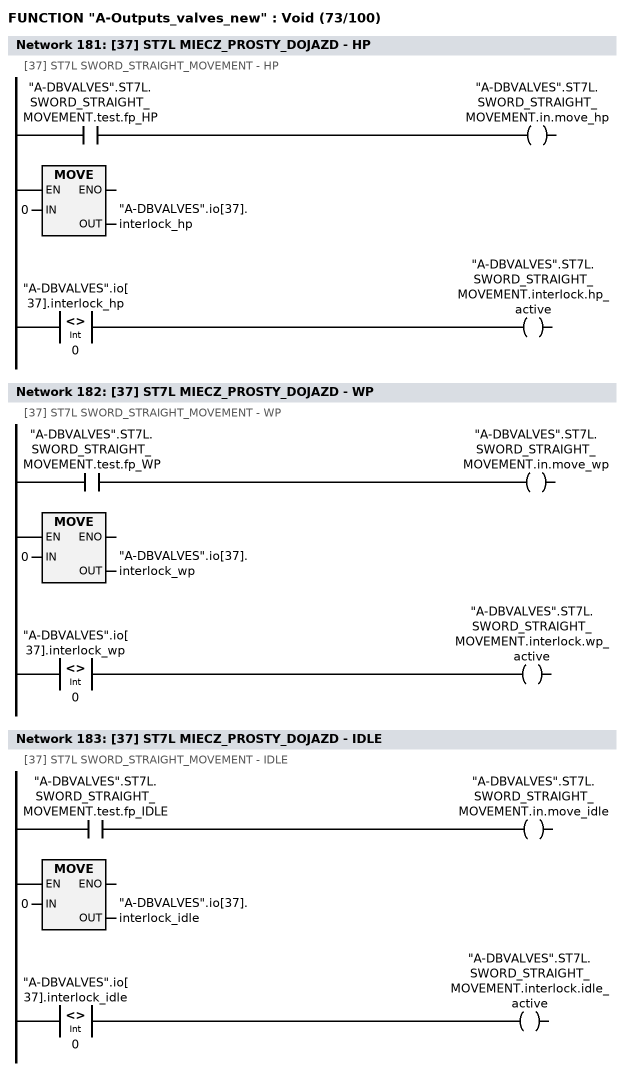
      O "A-DBVALVES".ST7L.SWORD_STRAIGHT_MOVEMENT.test.fp_HP;
//    O     "A-Flags".STATION.IN_HP_STEP
      = "A-DBVALVES".ST7L.SWORD_STRAIGHT_MOVEMENT.in.move_hp;

// Interlock hp
      L 0;
      T "A-DBVALVES".io[37].interlock_hp;

//{INTERLOCK_HP37}

      A(;
      L "A-DBVALVES".io[37].interlock_hp;
      L 0;
      <>I;
      );
      = "A-DBVALVES".ST7L.SWORD_STRAIGHT_MOVEMENT.interlock.hp_active;
NETWORK
TITLE = [37] ST7L MIECZ_PROSTY_DOJAZD - WP
//[37] ST7L SWORD_STRAIGHT_MOVEMENT - WP
      O "A-DBVALVES".ST7L.SWORD_STRAIGHT_MOVEMENT.test.fp_WP;
      = "A-DBVALVES".ST7L.SWORD_STRAIGHT_MOVEMENT.in.move_wp;

// Interlock wp
      L 0;
      T "A-DBVALVES".io[37].interlock_wp;

//{INTERLOCK_WP37}

      A(;
      L "A-DBVALVES".io[37].interlock_wp;
      L 0;
      <>I;
      );
      = "A-DBVALVES".ST7L.SWORD_STRAIGHT_MOVEMENT.interlock.wp_active;
NETWORK
TITLE = [37] ST7L MIECZ_PROSTY_DOJAZD - IDLE
//[37] ST7L SWORD_STRAIGHT_MOVEMENT - IDLE
      O "A-DBVALVES".ST7L.SWORD_STRAIGHT_MOVEMENT.test.fp_IDLE;
      = "A-DBVALVES".ST7L.SWORD_STRAIGHT_MOVEMENT.in.move_idle;

// Interlock idle
      L 0;
      T "A-DBVALVES".io[37].interlock_idle;

//{INTERLOCK_IDLE37}

      A(;
      L "A-DBVALVES".io[37].interlock_idle;
      L 0;
      <>I;
      );
      = "A-DBVALVES".ST7L.SWORD_STRAIGHT_MOVEMENT.interlock.idle_active;
NETWORK
TITLE = [37] ST7L MIECZ_PROSTY_DOJAZD
//[37] ST7L SWORD_STRAIGHT_MOVEMENT
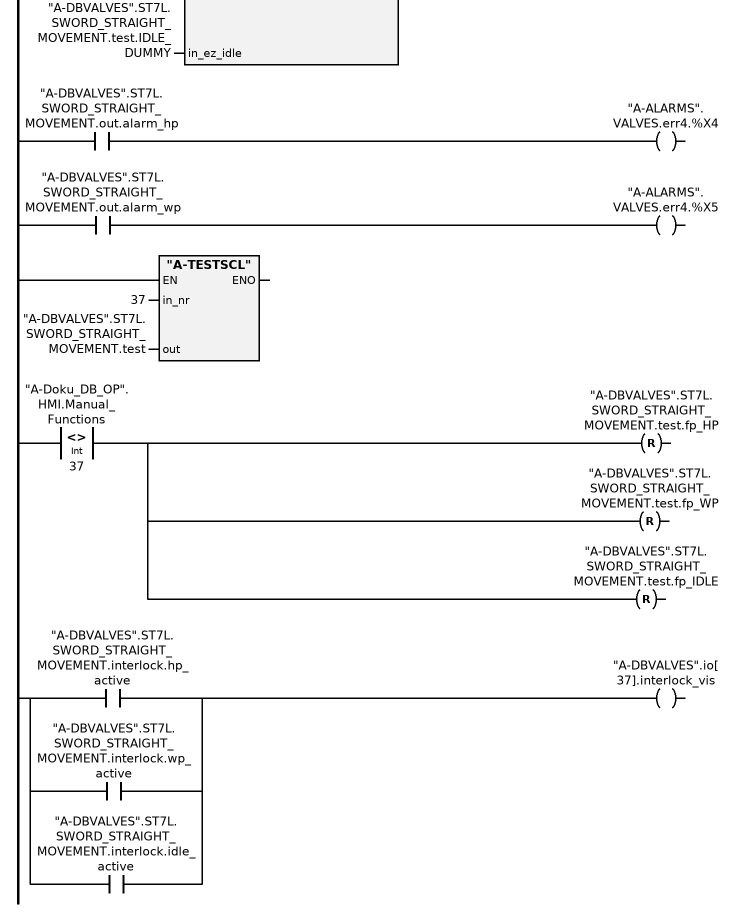
      CALL "3STATE_PISTON_with_brake", "INST_ST7L MIECZ_PROSTY_DOJAZD"
      (  in_safety_on                := "A-Flags".STATION.SAFETY_OK ,
         in_curtain_on               := "A-Flags".STATION.CURTAIN.OK ,
         in_move_hp                  := "A-DBVALVES".ST7L.SWORD_STRAIGHT_MOVEMENT.in.move_hp ,
         in_move_wp                  := "A-DBVALVES".ST7L.SWORD_STRAIGHT_MOVEMENT.in.move_wp ,
         in_move_idle                := "A-DBVALVES".ST7L.SWORD_STRAIGHT_MOVEMENT.in.move_idle ,
         in_interlock_hp             := "A-DBVALVES".ST7L.SWORD_STRAIGHT_MOVEMENT.interlock.hp_active ,
         in_interlock_wp             := "A-DBVALVES".ST7L.SWORD_STRAIGHT_MOVEMENT.interlock.wp_active ,
         in_interlock_idle           := "A-DBVALVES".ST7L.SWORD_STRAIGHT_MOVEMENT.interlock.idle_active ,
         in_sensor_hp1               := "ST7L-vsen_sword_straight_movement_HP_right" ,
         in_sensor_hp2               := "ST7L-vsen_sword_straight_movement_HP_right" ,
         in_sensor_wp1               := "ST7L-vsen_sword_straight_movement_WP_front" ,
         in_sensor_wp2               := "ST7L-vsen_sword_straight_movement_WP_front" ,
         out_in_hp                   := "A-DBVALVES".ST7L.SWORD_STRAIGHT_MOVEMENT.out.in_hp ,
         out_in_wp                   := "A-DBVALVES".ST7L.SWORD_STRAIGHT_MOVEMENT.out.in_wp ,
         out_idle                    := "A-DBVALVES".ST7L.SWORD_STRAIGHT_MOVEMENT.out.in_idle ,
         out_status                  := "A-DBVALVES".ST7L.SWORD_STRAIGHT_MOVEMENT.out.status ,
         out_brake                   := #brake ,
         out_alarm_hp                := "A-DBVALVES".ST7L.SWORD_STRAIGHT_MOVEMENT.out.alarm_hp ,
         out_alarm_wp                := "A-DBVALVES".ST7L.SWORD_STRAIGHT_MOVEMENT.out.alarm_wp ,
         out_alarm_idle              := "A-DBVALVES".ST7L.SWORD_STRAIGHT_MOVEMENT.out.alarm_idle ,
         out_diag_status             := "A-DBVALVES".ST7L.SWORD_STRAIGHT_MOVEMENT.out.diag_status ,
         out_interlock_show          := "A-DBVALVES".ST7L.SWORD_STRAIGHT_MOVEMENT.interlock.active ,
         in_ez_hp                    := "ST7L-ez_sword_straight_movement_HP_right" ,
         in_ez_wp                    := "ST7L-ez_sword_straight_movement_WP_front" ,
         in_ez_idle                  := "A-DBVALVES".ST7L.SWORD_STRAIGHT_MOVEMENT.test.IDLE_DUMMY
      );

      CALL "3STATE_DIAG"
      (  in_diag_status              := "A-DBVALVES".ST7L.SWORD_STRAIGHT_MOVEMENT.out.diag_status ,
         in_Ipw1                     := 'I120.0' ,
         in_Ipw2                     := ' ' ,
         in_Ipr1                     := 'I121.0' ,
         in_Ipr2                     := ' ' ,
         in_Qpw                      := 'Q3008.1' ,
         in_Qpr                      := 'Q3008.0' ,
         in_tio                      := "A-DBVALVES".io[37]
      );

      A "A-DBVALVES".ST7L.SWORD_STRAIGHT_MOVEMENT.out.alarm_hp;
      = "A-ALARMS".VALVES.err4.%X4;

      A "A-DBVALVES".ST7L.SWORD_STRAIGHT_MOVEMENT.out.alarm_wp;
      = "A-ALARMS".VALVES.err4.%X5;

      CALL "A-TESTSCL"
      (  in_nr                       := 37 ,
         out                         := "A-DBVALVES".ST7L.SWORD_STRAIGHT_MOVEMENT.test
      );

      A(;
      L "A-Doku_DB_OP".HMI.Manual_Functions;
      L 37;
      <>I;
      );
      R "A-DBVALVES".ST7L.SWORD_STRAIGHT_MOVEMENT.test.fp_HP;
      R "A-DBVALVES".ST7L.SWORD_STRAIGHT_MOVEMENT.test.fp_WP;
      R "A-DBVALVES".ST7L.SWORD_STRAIGHT_MOVEMENT.test.fp_IDLE;

      O "A-DBVALVES".ST7L.SWORD_STRAIGHT_MOVEMENT.interlock.hp_active;
      O "A-DBVALVES".ST7L.SWORD_STRAIGHT_MOVEMENT.interlock.wp_active;
      O "A-DBVALVES".ST7L.SWORD_STRAIGHT_MOVEMENT.interlock.idle_active;
      = "A-DBVALVES".io[37].interlock_vis;
NETWORK
TITLE = -

NETWORK
TITLE = [38] ST7L MIECZ_PROSTY - HP
//[38] ST7L SWORD_STRAIGHT - HP
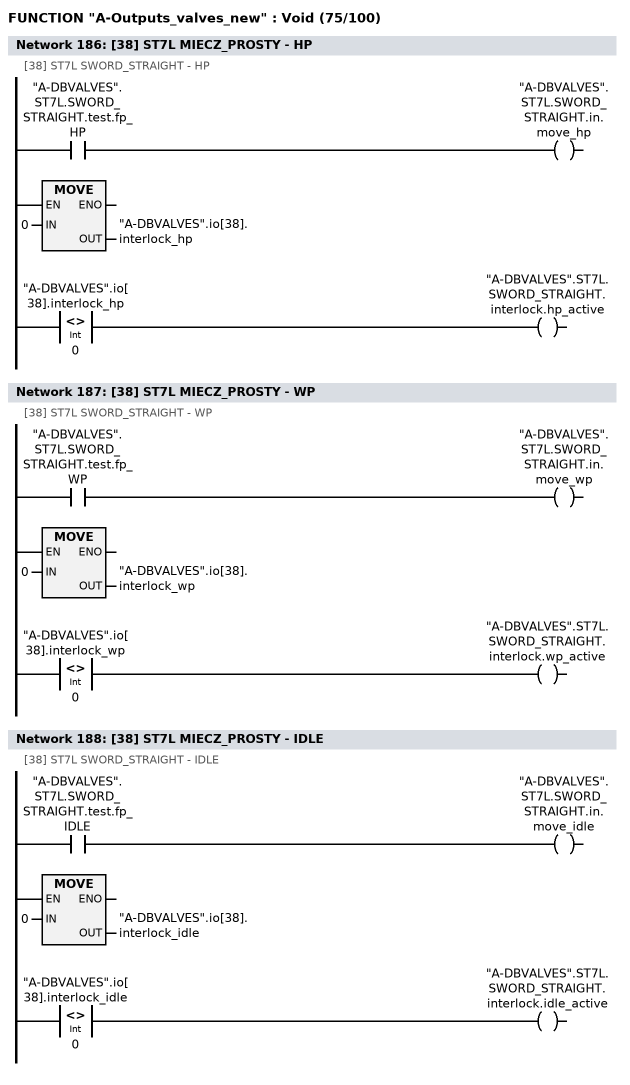
      O "A-DBVALVES".ST7L.SWORD_STRAIGHT.test.fp_HP;
//    O     "A-Flags".STATION.IN_HP_STEP
      = "A-DBVALVES".ST7L.SWORD_STRAIGHT.in.move_hp;

// Interlock hp
      L 0;
      T "A-DBVALVES".io[38].interlock_hp;

//{INTERLOCK_HP38}

      A(;
      L "A-DBVALVES".io[38].interlock_hp;
      L 0;
      <>I;
      );
      = "A-DBVALVES".ST7L.SWORD_STRAIGHT.interlock.hp_active;
NETWORK
TITLE = [38] ST7L MIECZ_PROSTY - WP
//[38] ST7L SWORD_STRAIGHT - WP
      O "A-DBVALVES".ST7L.SWORD_STRAIGHT.test.fp_WP;
      = "A-DBVALVES".ST7L.SWORD_STRAIGHT.in.move_wp;

// Interlock wp
      L 0;
      T "A-DBVALVES".io[38].interlock_wp;

//{INTERLOCK_WP38}

      A(;
      L "A-DBVALVES".io[38].interlock_wp;
      L 0;
      <>I;
      );
      = "A-DBVALVES".ST7L.SWORD_STRAIGHT.interlock.wp_active;
NETWORK
TITLE = [38] ST7L MIECZ_PROSTY - IDLE
//[38] ST7L SWORD_STRAIGHT - IDLE
      O "A-DBVALVES".ST7L.SWORD_STRAIGHT.test.fp_IDLE;
      = "A-DBVALVES".ST7L.SWORD_STRAIGHT.in.move_idle;

// Interlock idle
      L 0;
      T "A-DBVALVES".io[38].interlock_idle;

//{INTERLOCK_IDLE38}

      A(;
      L "A-DBVALVES".io[38].interlock_idle;
      L 0;
      <>I;
      );
      = "A-DBVALVES".ST7L.SWORD_STRAIGHT.interlock.idle_active;
NETWORK
TITLE = [38] ST7L MIECZ_PROSTY
//[38] ST7L SWORD_STRAIGHT
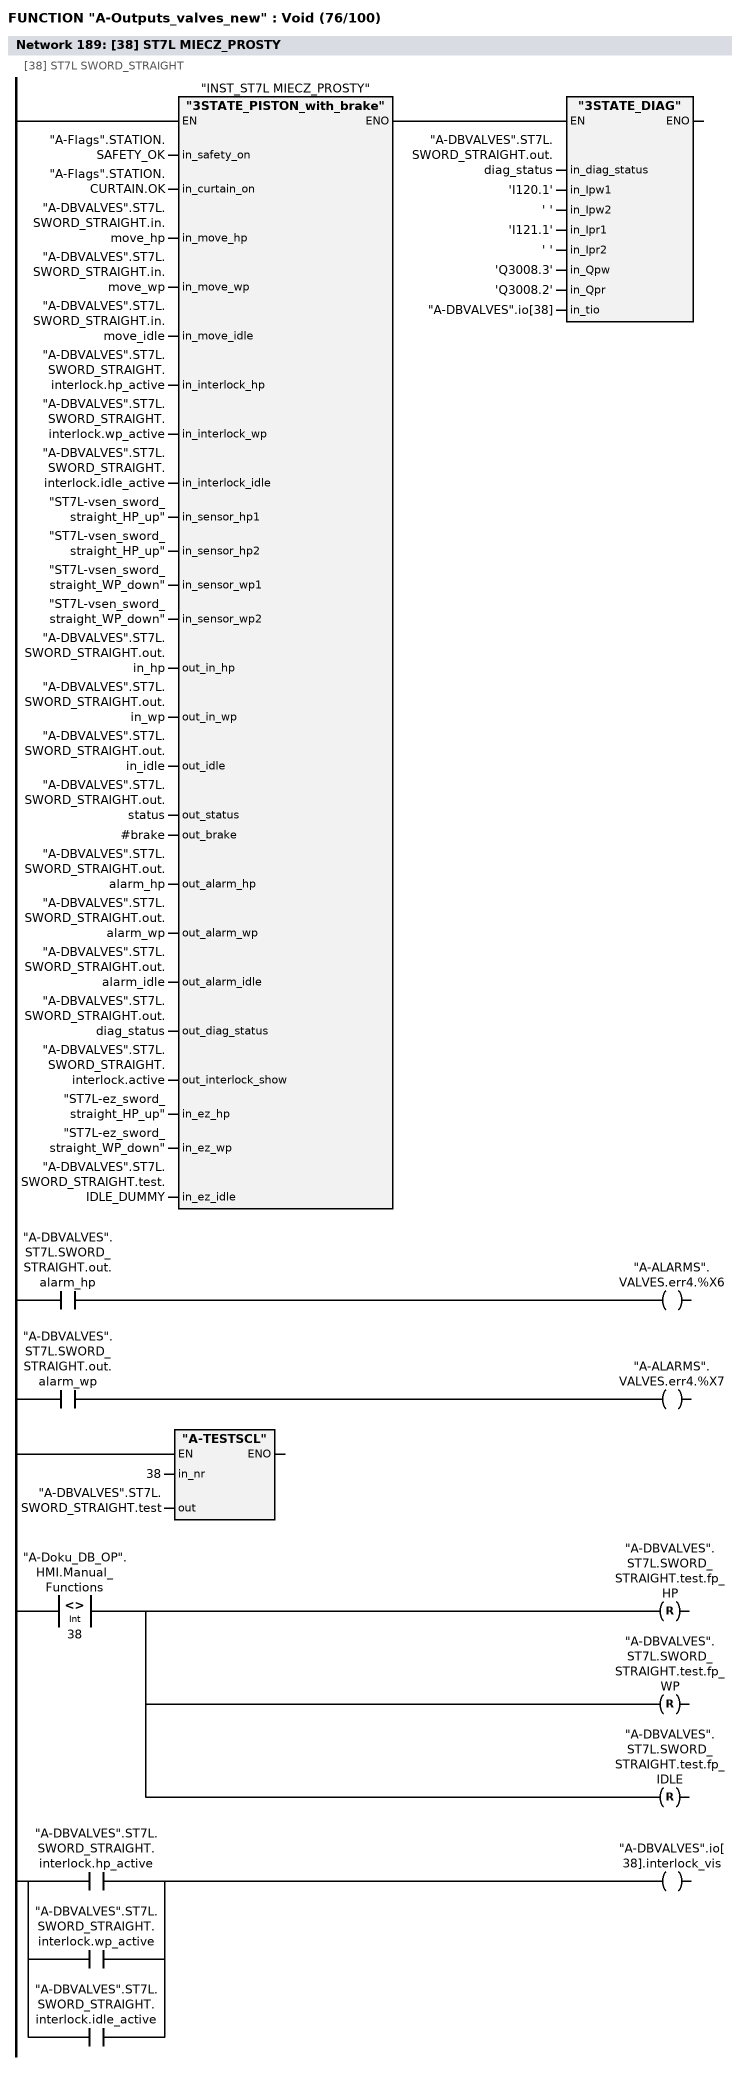
      CALL "3STATE_PISTON_with_brake", "INST_ST7L MIECZ_PROSTY"
      (  in_safety_on                := "A-Flags".STATION.SAFETY_OK ,
         in_curtain_on               := "A-Flags".STATION.CURTAIN.OK ,
         in_move_hp                  := "A-DBVALVES".ST7L.SWORD_STRAIGHT.in.move_hp ,
         in_move_wp                  := "A-DBVALVES".ST7L.SWORD_STRAIGHT.in.move_wp ,
         in_move_idle                := "A-DBVALVES".ST7L.SWORD_STRAIGHT.in.move_idle ,
         in_interlock_hp             := "A-DBVALVES".ST7L.SWORD_STRAIGHT.interlock.hp_active ,
         in_interlock_wp             := "A-DBVALVES".ST7L.SWORD_STRAIGHT.interlock.wp_active ,
         in_interlock_idle           := "A-DBVALVES".ST7L.SWORD_STRAIGHT.interlock.idle_active ,
         in_sensor_hp1               := "ST7L-vsen_sword_straight_HP_up" ,
         in_sensor_hp2               := "ST7L-vsen_sword_straight_HP_up" ,
         in_sensor_wp1               := "ST7L-vsen_sword_straight_WP_down" ,
         in_sensor_wp2               := "ST7L-vsen_sword_straight_WP_down" ,
         out_in_hp                   := "A-DBVALVES".ST7L.SWORD_STRAIGHT.out.in_hp ,
         out_in_wp                   := "A-DBVALVES".ST7L.SWORD_STRAIGHT.out.in_wp ,
         out_idle                    := "A-DBVALVES".ST7L.SWORD_STRAIGHT.out.in_idle ,
         out_status                  := "A-DBVALVES".ST7L.SWORD_STRAIGHT.out.status ,
         out_brake                   := #brake ,
         out_alarm_hp                := "A-DBVALVES".ST7L.SWORD_STRAIGHT.out.alarm_hp ,
         out_alarm_wp                := "A-DBVALVES".ST7L.SWORD_STRAIGHT.out.alarm_wp ,
         out_alarm_idle              := "A-DBVALVES".ST7L.SWORD_STRAIGHT.out.alarm_idle ,
         out_diag_status             := "A-DBVALVES".ST7L.SWORD_STRAIGHT.out.diag_status ,
         out_interlock_show          := "A-DBVALVES".ST7L.SWORD_STRAIGHT.interlock.active ,
         in_ez_hp                    := "ST7L-ez_sword_straight_HP_up" ,
         in_ez_wp                    := "ST7L-ez_sword_straight_WP_down" ,
         in_ez_idle                  := "A-DBVALVES".ST7L.SWORD_STRAIGHT.test.IDLE_DUMMY
      );

      CALL "3STATE_DIAG"
      (  in_diag_status              := "A-DBVALVES".ST7L.SWORD_STRAIGHT.out.diag_status ,
         in_Ipw1                     := 'I120.1' ,
         in_Ipw2                     := ' ' ,
         in_Ipr1                     := 'I121.1' ,
         in_Ipr2                     := ' ' ,
         in_Qpw                      := 'Q3008.3' ,
         in_Qpr                      := 'Q3008.2' ,
         in_tio                      := "A-DBVALVES".io[38]
      );

      A "A-DBVALVES".ST7L.SWORD_STRAIGHT.out.alarm_hp;
      = "A-ALARMS".VALVES.err4.%X6;

      A "A-DBVALVES".ST7L.SWORD_STRAIGHT.out.alarm_wp;
      = "A-ALARMS".VALVES.err4.%X7;

      CALL "A-TESTSCL"
      (  in_nr                       := 38 ,
         out                         := "A-DBVALVES".ST7L.SWORD_STRAIGHT.test
      );

      A(;
      L "A-Doku_DB_OP".HMI.Manual_Functions;
      L 38;
      <>I;
      );
      R "A-DBVALVES".ST7L.SWORD_STRAIGHT.test.fp_HP;
      R "A-DBVALVES".ST7L.SWORD_STRAIGHT.test.fp_WP;
      R "A-DBVALVES".ST7L.SWORD_STRAIGHT.test.fp_IDLE;

      O "A-DBVALVES".ST7L.SWORD_STRAIGHT.interlock.hp_active;
      O "A-DBVALVES".ST7L.SWORD_STRAIGHT.interlock.wp_active;
      O "A-DBVALVES".ST7L.SWORD_STRAIGHT.interlock.idle_active;
      = "A-DBVALVES".io[38].interlock_vis;
NETWORK
TITLE = -

NETWORK
TITLE = [39] ST7L MIECZ_RUCHOMY_DOJAZD - HP
//[39] ST7L SWORD_MOBILE_MOVEMENT - HP
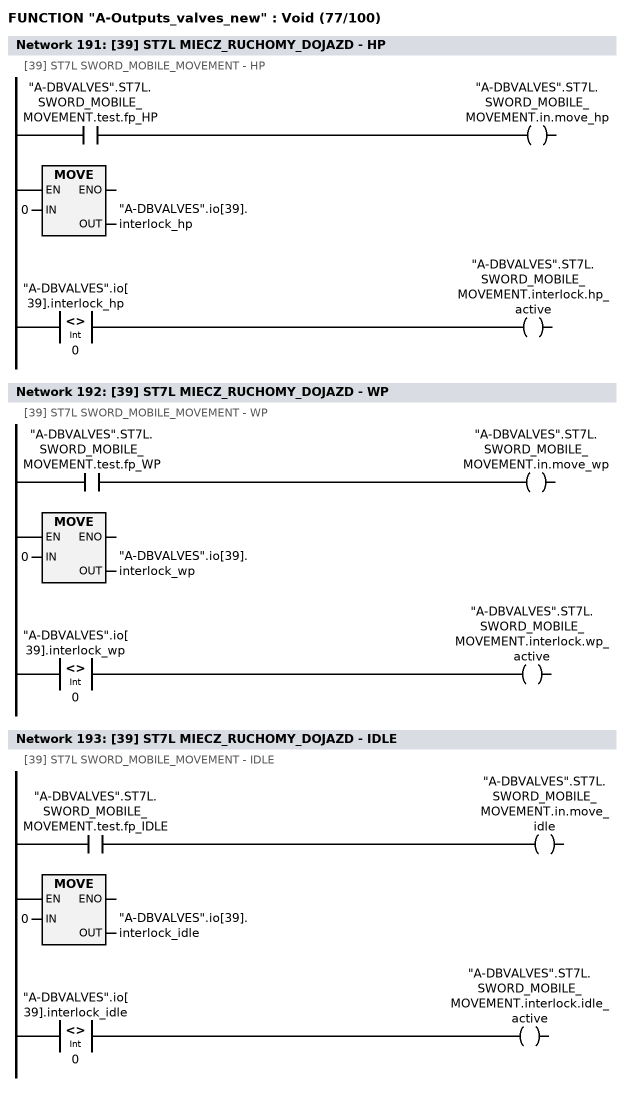
      O "A-DBVALVES".ST7L.SWORD_MOBILE_MOVEMENT.test.fp_HP;
//    O     "A-Flags".STATION.IN_HP_STEP
      = "A-DBVALVES".ST7L.SWORD_MOBILE_MOVEMENT.in.move_hp;

// Interlock hp
      L 0;
      T "A-DBVALVES".io[39].interlock_hp;

//{INTERLOCK_HP39}

      A(;
      L "A-DBVALVES".io[39].interlock_hp;
      L 0;
      <>I;
      );
      = "A-DBVALVES".ST7L.SWORD_MOBILE_MOVEMENT.interlock.hp_active;
NETWORK
TITLE = [39] ST7L MIECZ_RUCHOMY_DOJAZD - WP
//[39] ST7L SWORD_MOBILE_MOVEMENT - WP
      O "A-DBVALVES".ST7L.SWORD_MOBILE_MOVEMENT.test.fp_WP;
      = "A-DBVALVES".ST7L.SWORD_MOBILE_MOVEMENT.in.move_wp;

// Interlock wp
      L 0;
      T "A-DBVALVES".io[39].interlock_wp;

//{INTERLOCK_WP39}

      A(;
      L "A-DBVALVES".io[39].interlock_wp;
      L 0;
      <>I;
      );
      = "A-DBVALVES".ST7L.SWORD_MOBILE_MOVEMENT.interlock.wp_active;
NETWORK
TITLE = [39] ST7L MIECZ_RUCHOMY_DOJAZD - IDLE
//[39] ST7L SWORD_MOBILE_MOVEMENT - IDLE
      O "A-DBVALVES".ST7L.SWORD_MOBILE_MOVEMENT.test.fp_IDLE;
      = "A-DBVALVES".ST7L.SWORD_MOBILE_MOVEMENT.in.move_idle;

// Interlock idle
      L 0;
      T "A-DBVALVES".io[39].interlock_idle;

//{INTERLOCK_IDLE39}

      A(;
      L "A-DBVALVES".io[39].interlock_idle;
      L 0;
      <>I;
      );
      = "A-DBVALVES".ST7L.SWORD_MOBILE_MOVEMENT.interlock.idle_active;
NETWORK
TITLE = [39] ST7L MIECZ_RUCHOMY_DOJAZD
//[39] ST7L SWORD_MOBILE_MOVEMENT
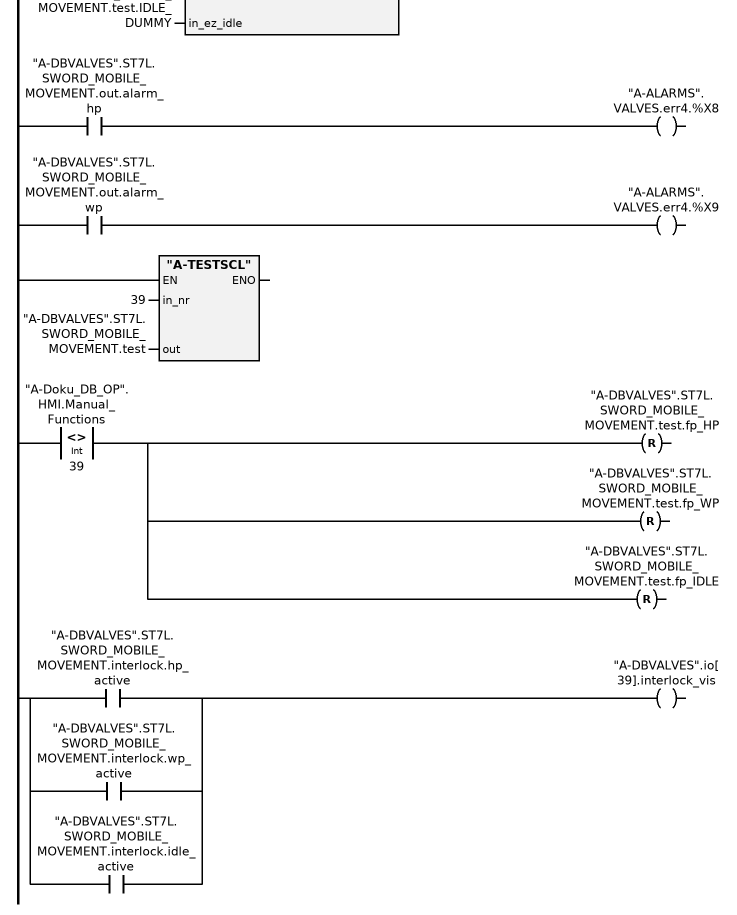
      CALL "3STATE_PISTON_with_brake", "INST_ST7L MIECZ_RUCHOMY_DOJAZD"
      (  in_safety_on                := "A-Flags".STATION.SAFETY_OK ,
         in_curtain_on               := "A-Flags".STATION.CURTAIN.OK ,
         in_move_hp                  := "A-DBVALVES".ST7L.SWORD_MOBILE_MOVEMENT.in.move_hp ,
         in_move_wp                  := "A-DBVALVES".ST7L.SWORD_MOBILE_MOVEMENT.in.move_wp ,
         in_move_idle                := "A-DBVALVES".ST7L.SWORD_MOBILE_MOVEMENT.in.move_idle ,
         in_interlock_hp             := "A-DBVALVES".ST7L.SWORD_MOBILE_MOVEMENT.interlock.hp_active ,
         in_interlock_wp             := "A-DBVALVES".ST7L.SWORD_MOBILE_MOVEMENT.interlock.wp_active ,
         in_interlock_idle           := "A-DBVALVES".ST7L.SWORD_MOBILE_MOVEMENT.interlock.idle_active ,
         in_sensor_hp1               := "ST7L-vsen_sword_mobile_movement_HP_right" ,
         in_sensor_hp2               := "ST7L-vsen_sword_mobile_movement_HP_right" ,
         in_sensor_wp1               := "ST7L-vsen_sword_mobile_movement_WP_front" ,
         in_sensor_wp2               := "ST7L-vsen_sword_mobile_movement_WP_front" ,
         out_in_hp                   := "A-DBVALVES".ST7L.SWORD_MOBILE_MOVEMENT.out.in_hp ,
         out_in_wp                   := "A-DBVALVES".ST7L.SWORD_MOBILE_MOVEMENT.out.in_wp ,
         out_idle                    := "A-DBVALVES".ST7L.SWORD_MOBILE_MOVEMENT.out.in_idle ,
         out_status                  := "A-DBVALVES".ST7L.SWORD_MOBILE_MOVEMENT.out.status ,
         out_brake                   := #brake ,
         out_alarm_hp                := "A-DBVALVES".ST7L.SWORD_MOBILE_MOVEMENT.out.alarm_hp ,
         out_alarm_wp                := "A-DBVALVES".ST7L.SWORD_MOBILE_MOVEMENT.out.alarm_wp ,
         out_alarm_idle              := "A-DBVALVES".ST7L.SWORD_MOBILE_MOVEMENT.out.alarm_idle ,
         out_diag_status             := "A-DBVALVES".ST7L.SWORD_MOBILE_MOVEMENT.out.diag_status ,
         out_interlock_show          := "A-DBVALVES".ST7L.SWORD_MOBILE_MOVEMENT.interlock.active ,
         in_ez_hp                    := "ST7L-ez_sword_mobile_movement_HP_right" ,
         in_ez_wp                    := "ST7L-ez_sword_mobile_movement_WP_front" ,
         in_ez_idle                  := "A-DBVALVES".ST7L.SWORD_MOBILE_MOVEMENT.test.IDLE_DUMMY
      );

      CALL "3STATE_DIAG"
      (  in_diag_status              := "A-DBVALVES".ST7L.SWORD_MOBILE_MOVEMENT.out.diag_status ,
         in_Ipw1                     := 'I120.3' ,
         in_Ipw2                     := ' ' ,
         in_Ipr1                     := 'I121.3' ,
         in_Ipr2                     := ' ' ,
         in_Qpw                      := 'Q3008.7' ,
         in_Qpr                      := 'Q3008.6' ,
         in_tio                      := "A-DBVALVES".io[39]
      );

      A "A-DBVALVES".ST7L.SWORD_MOBILE_MOVEMENT.out.alarm_hp;
      = "A-ALARMS".VALVES.err4.%X8;

      A "A-DBVALVES".ST7L.SWORD_MOBILE_MOVEMENT.out.alarm_wp;
      = "A-ALARMS".VALVES.err4.%X9;

      CALL "A-TESTSCL"
      (  in_nr                       := 39 ,
         out                         := "A-DBVALVES".ST7L.SWORD_MOBILE_MOVEMENT.test
      );

      A(;
      L "A-Doku_DB_OP".HMI.Manual_Functions;
      L 39;
      <>I;
      );
      R "A-DBVALVES".ST7L.SWORD_MOBILE_MOVEMENT.test.fp_HP;
      R "A-DBVALVES".ST7L.SWORD_MOBILE_MOVEMENT.test.fp_WP;
      R "A-DBVALVES".ST7L.SWORD_MOBILE_MOVEMENT.test.fp_IDLE;

      O "A-DBVALVES".ST7L.SWORD_MOBILE_MOVEMENT.interlock.hp_active;
      O "A-DBVALVES".ST7L.SWORD_MOBILE_MOVEMENT.interlock.wp_active;
      O "A-DBVALVES".ST7L.SWORD_MOBILE_MOVEMENT.interlock.idle_active;
      = "A-DBVALVES".io[39].interlock_vis;
NETWORK
TITLE = -

NETWORK
TITLE = [40] ST7L MIECZ_RUCHOMY_PRZEJAZD - HP
//[40] ST7L SWORD_MOBILE_SLIDE - HP
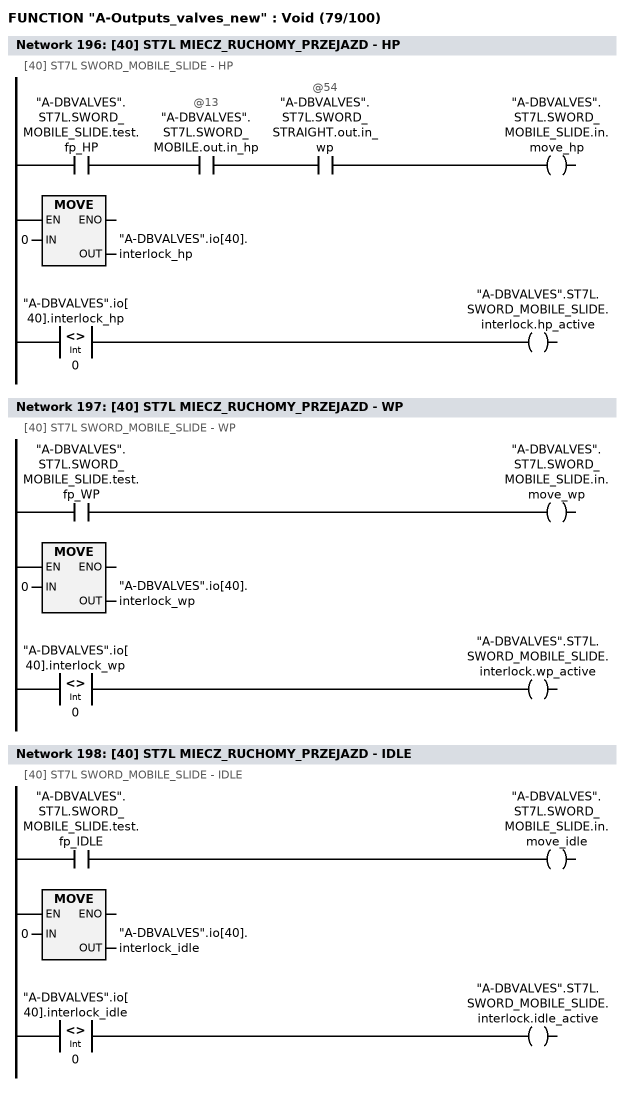
      O "A-DBVALVES".ST7L.SWORD_MOBILE_SLIDE.test.fp_HP;
//    O     "A-Flags".STATION.IN_HP_STEP
      A "A-DBVALVES".ST7L.SWORD_MOBILE.out.in_hp;// @13
      A "A-DBVALVES".ST7L.SWORD_STRAIGHT.out.in_wp;// @54
      = "A-DBVALVES".ST7L.SWORD_MOBILE_SLIDE.in.move_hp;

// Interlock hp
      L 0;
      T "A-DBVALVES".io[40].interlock_hp;

//{INTERLOCK_HP40}

      A(;
      L "A-DBVALVES".io[40].interlock_hp;
      L 0;
      <>I;
      );
      = "A-DBVALVES".ST7L.SWORD_MOBILE_SLIDE.interlock.hp_active;
NETWORK
TITLE = [40] ST7L MIECZ_RUCHOMY_PRZEJAZD - WP
//[40] ST7L SWORD_MOBILE_SLIDE - WP
      O "A-DBVALVES".ST7L.SWORD_MOBILE_SLIDE.test.fp_WP;
      = "A-DBVALVES".ST7L.SWORD_MOBILE_SLIDE.in.move_wp;

// Interlock wp
      L 0;
      T "A-DBVALVES".io[40].interlock_wp;

//{INTERLOCK_WP40}

      A(;
      L "A-DBVALVES".io[40].interlock_wp;
      L 0;
      <>I;
      );
      = "A-DBVALVES".ST7L.SWORD_MOBILE_SLIDE.interlock.wp_active;
NETWORK
TITLE = [40] ST7L MIECZ_RUCHOMY_PRZEJAZD - IDLE
//[40] ST7L SWORD_MOBILE_SLIDE - IDLE
      O "A-DBVALVES".ST7L.SWORD_MOBILE_SLIDE.test.fp_IDLE;
      = "A-DBVALVES".ST7L.SWORD_MOBILE_SLIDE.in.move_idle;

// Interlock idle
      L 0;
      T "A-DBVALVES".io[40].interlock_idle;

//{INTERLOCK_IDLE40}

      A(;
      L "A-DBVALVES".io[40].interlock_idle;
      L 0;
      <>I;
      );
      = "A-DBVALVES".ST7L.SWORD_MOBILE_SLIDE.interlock.idle_active;
NETWORK
TITLE = [40] ST7L MIECZ_RUCHOMY_PRZEJAZD
//[40] ST7L SWORD_MOBILE_SLIDE
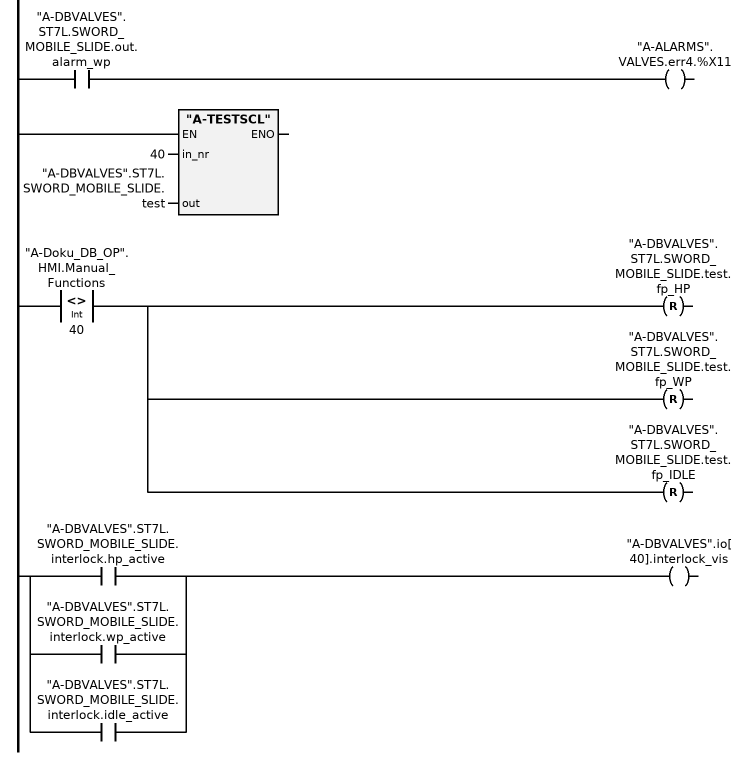
      CALL "3STATE_PISTON_with_brake", "INST_ST7L MIECZ_RUCHOMY_PRZEJAZD"
      (  in_safety_on                := "A-Flags".STATION.SAFETY_OK ,
         in_curtain_on               := "A-Flags".STATION.CURTAIN.OK ,
         in_move_hp                  := "A-DBVALVES".ST7L.SWORD_MOBILE_SLIDE.in.move_hp ,
         in_move_wp                  := "A-DBVALVES".ST7L.SWORD_MOBILE_SLIDE.in.move_wp ,
         in_move_idle                := "A-DBVALVES".ST7L.SWORD_MOBILE_SLIDE.in.move_idle ,
         in_interlock_hp             := "A-DBVALVES".ST7L.SWORD_MOBILE_SLIDE.interlock.hp_active ,
         in_interlock_wp             := "A-DBVALVES".ST7L.SWORD_MOBILE_SLIDE.interlock.wp_active ,
         in_interlock_idle           := "A-DBVALVES".ST7L.SWORD_MOBILE_SLIDE.interlock.idle_active ,
         in_sensor_hp1               := "ST7L-vsen_sword_mobile_slide_HP_left" ,
         in_sensor_hp2               := "ST7L-vsen_sword_mobile_slide_HP_left" ,
         in_sensor_wp1               := "ST7L-vsen_sword_mobile_slide_WP_right" ,
         in_sensor_wp2               := "ST7L-vsen_sword_mobile_slide_WP_right" ,
         out_in_hp                   := "A-DBVALVES".ST7L.SWORD_MOBILE_SLIDE.out.in_hp ,
         out_in_wp                   := "A-DBVALVES".ST7L.SWORD_MOBILE_SLIDE.out.in_wp ,
         out_idle                    := "A-DBVALVES".ST7L.SWORD_MOBILE_SLIDE.out.in_idle ,
         out_status                  := "A-DBVALVES".ST7L.SWORD_MOBILE_SLIDE.out.status ,
         out_brake                   := #brake ,
         out_alarm_hp                := "A-DBVALVES".ST7L.SWORD_MOBILE_SLIDE.out.alarm_hp ,
         out_alarm_wp                := "A-DBVALVES".ST7L.SWORD_MOBILE_SLIDE.out.alarm_wp ,
         out_alarm_idle              := "A-DBVALVES".ST7L.SWORD_MOBILE_SLIDE.out.alarm_idle ,
         out_diag_status             := "A-DBVALVES".ST7L.SWORD_MOBILE_SLIDE.out.diag_status ,
         out_interlock_show          := "A-DBVALVES".ST7L.SWORD_MOBILE_SLIDE.interlock.active ,
         in_ez_hp                    := "ST7L-ez_sword_mobile_slide_HP_left" ,
         in_ez_wp                    := "ST7L-ez_sword_mobile_slide_WP_right" ,
         in_ez_idle                  := "A-DBVALVES".ST7L.SWORD_MOBILE_SLIDE.test.IDLE_DUMMY
      );

      CALL "3STATE_DIAG"
      (  in_diag_status              := "A-DBVALVES".ST7L.SWORD_MOBILE_SLIDE.out.diag_status ,
         in_Ipw1                     := 'I120.2' ,
         in_Ipw2                     := ' ' ,
         in_Ipr1                     := 'I121.2' ,
         in_Ipr2                     := ' ' ,
         in_Qpw                      := 'Q3008.5' ,
         in_Qpr                      := 'Q3008.4' ,
         in_tio                      := "A-DBVALVES".io[40]
      );

      A "A-DBVALVES".ST7L.SWORD_MOBILE_SLIDE.out.alarm_hp;
      = "A-ALARMS".VALVES.err4.%X10;

      A "A-DBVALVES".ST7L.SWORD_MOBILE_SLIDE.out.alarm_wp;
      = "A-ALARMS".VALVES.err4.%X11;

      CALL "A-TESTSCL"
      (  in_nr                       := 40 ,
         out                         := "A-DBVALVES".ST7L.SWORD_MOBILE_SLIDE.test
      );

      A(;
      L "A-Doku_DB_OP".HMI.Manual_Functions;
      L 40;
      <>I;
      );
      R "A-DBVALVES".ST7L.SWORD_MOBILE_SLIDE.test.fp_HP;
      R "A-DBVALVES".ST7L.SWORD_MOBILE_SLIDE.test.fp_WP;
      R "A-DBVALVES".ST7L.SWORD_MOBILE_SLIDE.test.fp_IDLE;

      O "A-DBVALVES".ST7L.SWORD_MOBILE_SLIDE.interlock.hp_active;
      O "A-DBVALVES".ST7L.SWORD_MOBILE_SLIDE.interlock.wp_active;
      O "A-DBVALVES".ST7L.SWORD_MOBILE_SLIDE.interlock.idle_active;
      = "A-DBVALVES".io[40].interlock_vis;
NETWORK
TITLE = -

NETWORK
TITLE = [41] ST7L MIECZ_RUCHOMY - HP
//[41] ST7L SWORD_MOBILE - HP
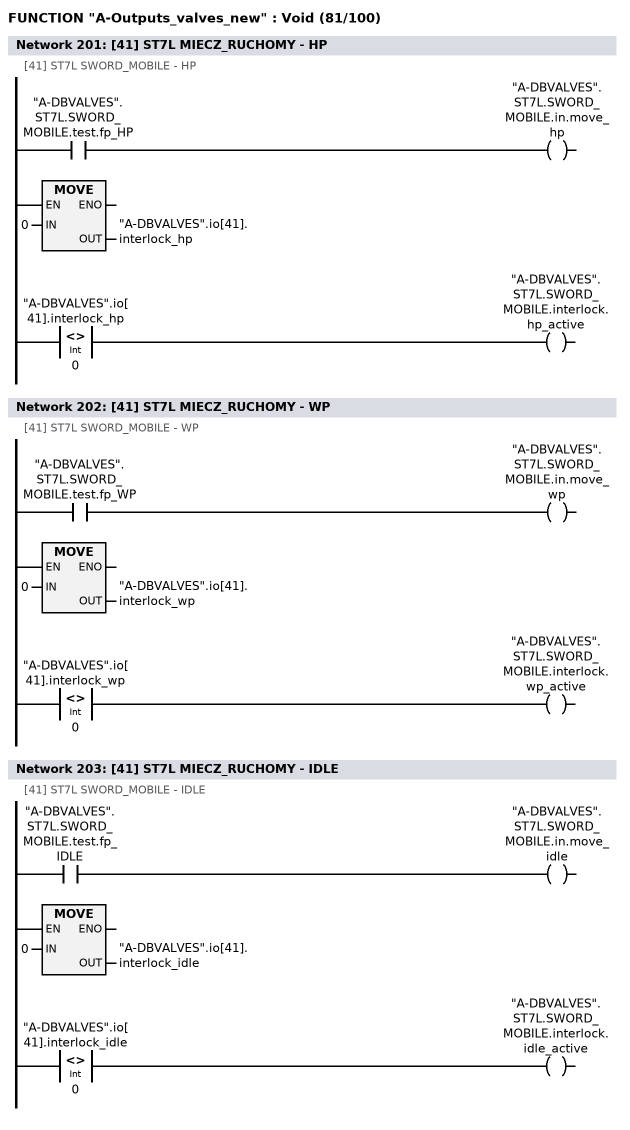
      O "A-DBVALVES".ST7L.SWORD_MOBILE.test.fp_HP;
//    O     "A-Flags".STATION.IN_HP_STEP
      = "A-DBVALVES".ST7L.SWORD_MOBILE.in.move_hp;

// Interlock hp
      L 0;
      T "A-DBVALVES".io[41].interlock_hp;

//{INTERLOCK_HP41}

      A(;
      L "A-DBVALVES".io[41].interlock_hp;
      L 0;
      <>I;
      );
      = "A-DBVALVES".ST7L.SWORD_MOBILE.interlock.hp_active;
NETWORK
TITLE = [41] ST7L MIECZ_RUCHOMY - WP
//[41] ST7L SWORD_MOBILE - WP
      O "A-DBVALVES".ST7L.SWORD_MOBILE.test.fp_WP;
      = "A-DBVALVES".ST7L.SWORD_MOBILE.in.move_wp;

// Interlock wp
      L 0;
      T "A-DBVALVES".io[41].interlock_wp;

//{INTERLOCK_WP41}

      A(;
      L "A-DBVALVES".io[41].interlock_wp;
      L 0;
      <>I;
      );
      = "A-DBVALVES".ST7L.SWORD_MOBILE.interlock.wp_active;
NETWORK
TITLE = [41] ST7L MIECZ_RUCHOMY - IDLE
//[41] ST7L SWORD_MOBILE - IDLE
      O "A-DBVALVES".ST7L.SWORD_MOBILE.test.fp_IDLE;
      = "A-DBVALVES".ST7L.SWORD_MOBILE.in.move_idle;

// Interlock idle
      L 0;
      T "A-DBVALVES".io[41].interlock_idle;

//{INTERLOCK_IDLE41}

      A(;
      L "A-DBVALVES".io[41].interlock_idle;
      L 0;
      <>I;
      );
      = "A-DBVALVES".ST7L.SWORD_MOBILE.interlock.idle_active;
NETWORK
TITLE = [41] ST7L MIECZ_RUCHOMY
//[41] ST7L SWORD_MOBILE
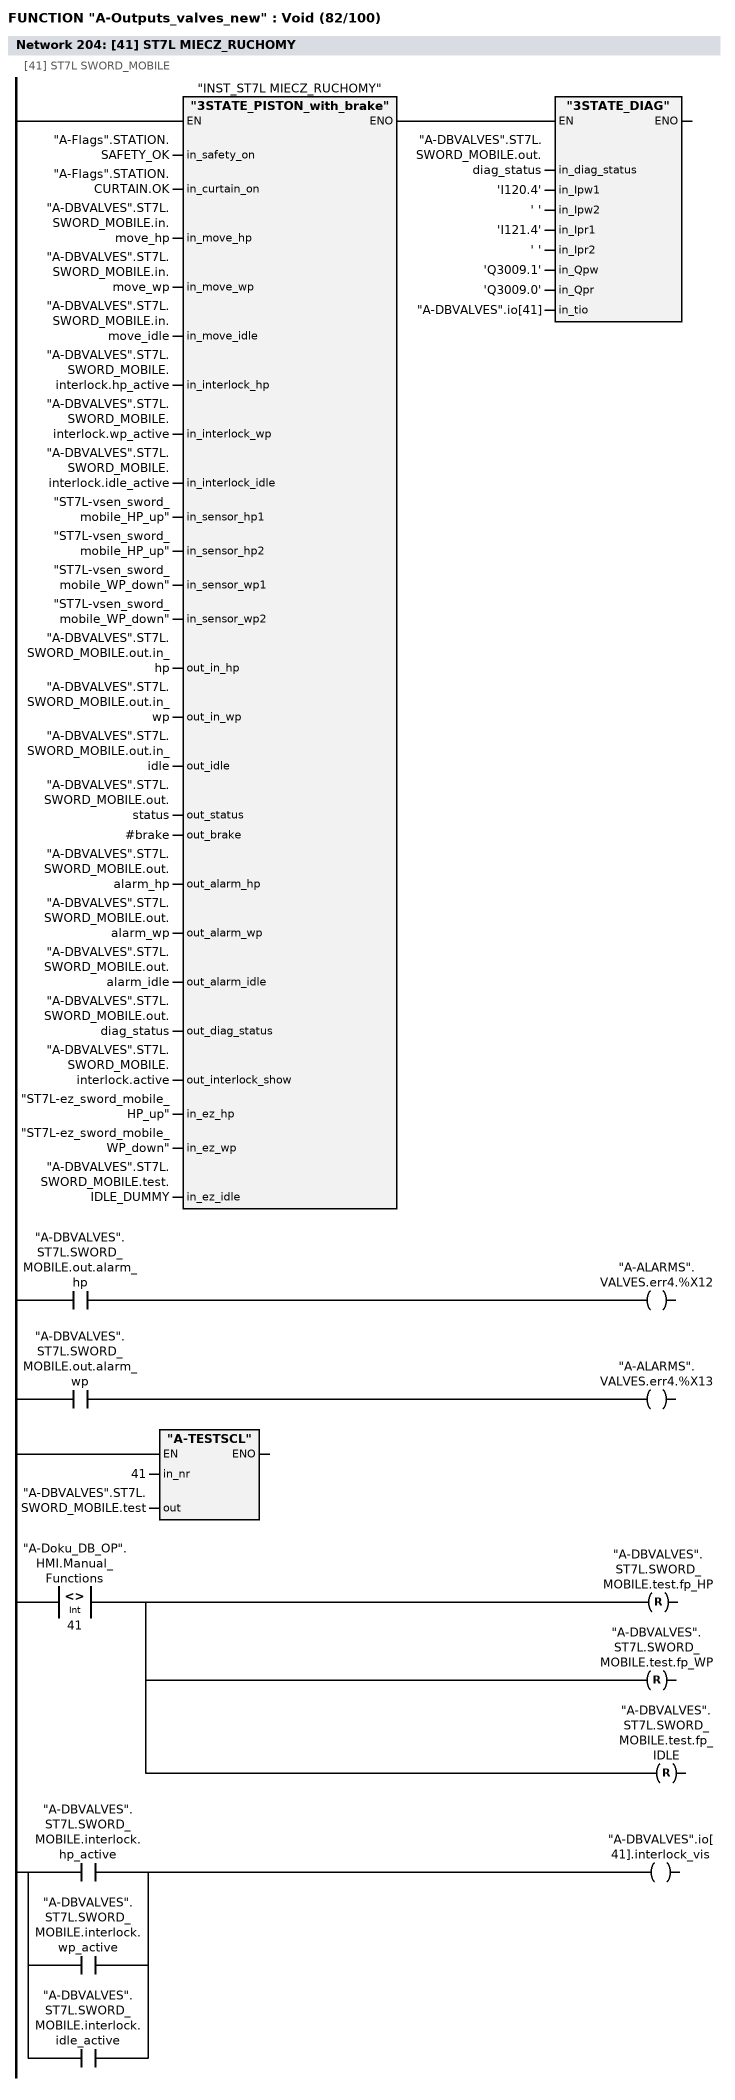
      CALL "3STATE_PISTON_with_brake", "INST_ST7L MIECZ_RUCHOMY"
      (  in_safety_on                := "A-Flags".STATION.SAFETY_OK ,
         in_curtain_on               := "A-Flags".STATION.CURTAIN.OK ,
         in_move_hp                  := "A-DBVALVES".ST7L.SWORD_MOBILE.in.move_hp ,
         in_move_wp                  := "A-DBVALVES".ST7L.SWORD_MOBILE.in.move_wp ,
         in_move_idle                := "A-DBVALVES".ST7L.SWORD_MOBILE.in.move_idle ,
         in_interlock_hp             := "A-DBVALVES".ST7L.SWORD_MOBILE.interlock.hp_active ,
         in_interlock_wp             := "A-DBVALVES".ST7L.SWORD_MOBILE.interlock.wp_active ,
         in_interlock_idle           := "A-DBVALVES".ST7L.SWORD_MOBILE.interlock.idle_active ,
         in_sensor_hp1               := "ST7L-vsen_sword_mobile_HP_up" ,
         in_sensor_hp2               := "ST7L-vsen_sword_mobile_HP_up" ,
         in_sensor_wp1               := "ST7L-vsen_sword_mobile_WP_down" ,
         in_sensor_wp2               := "ST7L-vsen_sword_mobile_WP_down" ,
         out_in_hp                   := "A-DBVALVES".ST7L.SWORD_MOBILE.out.in_hp ,
         out_in_wp                   := "A-DBVALVES".ST7L.SWORD_MOBILE.out.in_wp ,
         out_idle                    := "A-DBVALVES".ST7L.SWORD_MOBILE.out.in_idle ,
         out_status                  := "A-DBVALVES".ST7L.SWORD_MOBILE.out.status ,
         out_brake                   := #brake ,
         out_alarm_hp                := "A-DBVALVES".ST7L.SWORD_MOBILE.out.alarm_hp ,
         out_alarm_wp                := "A-DBVALVES".ST7L.SWORD_MOBILE.out.alarm_wp ,
         out_alarm_idle              := "A-DBVALVES".ST7L.SWORD_MOBILE.out.alarm_idle ,
         out_diag_status             := "A-DBVALVES".ST7L.SWORD_MOBILE.out.diag_status ,
         out_interlock_show          := "A-DBVALVES".ST7L.SWORD_MOBILE.interlock.active ,
         in_ez_hp                    := "ST7L-ez_sword_mobile_HP_up" ,
         in_ez_wp                    := "ST7L-ez_sword_mobile_WP_down" ,
         in_ez_idle                  := "A-DBVALVES".ST7L.SWORD_MOBILE.test.IDLE_DUMMY
      );

      CALL "3STATE_DIAG"
      (  in_diag_status              := "A-DBVALVES".ST7L.SWORD_MOBILE.out.diag_status ,
         in_Ipw1                     := 'I120.4' ,
         in_Ipw2                     := ' ' ,
         in_Ipr1                     := 'I121.4' ,
         in_Ipr2                     := ' ' ,
         in_Qpw                      := 'Q3009.1' ,
         in_Qpr                      := 'Q3009.0' ,
         in_tio                      := "A-DBVALVES".io[41]
      );

      A "A-DBVALVES".ST7L.SWORD_MOBILE.out.alarm_hp;
      = "A-ALARMS".VALVES.err4.%X12;

      A "A-DBVALVES".ST7L.SWORD_MOBILE.out.alarm_wp;
      = "A-ALARMS".VALVES.err4.%X13;

      CALL "A-TESTSCL"
      (  in_nr                       := 41 ,
         out                         := "A-DBVALVES".ST7L.SWORD_MOBILE.test
      );

      A(;
      L "A-Doku_DB_OP".HMI.Manual_Functions;
      L 41;
      <>I;
      );
      R "A-DBVALVES".ST7L.SWORD_MOBILE.test.fp_HP;
      R "A-DBVALVES".ST7L.SWORD_MOBILE.test.fp_WP;
      R "A-DBVALVES".ST7L.SWORD_MOBILE.test.fp_IDLE;

      O "A-DBVALVES".ST7L.SWORD_MOBILE.interlock.hp_active;
      O "A-DBVALVES".ST7L.SWORD_MOBILE.interlock.wp_active;
      O "A-DBVALVES".ST7L.SWORD_MOBILE.interlock.idle_active;
      = "A-DBVALVES".io[41].interlock_vis;
NETWORK
TITLE = -

NETWORK
TITLE = [42] ST7R MIECZ_SKOSNY_DOJAZD - HP
//[42] ST7R SWORD_ANGLE_MOVEMENT - HP
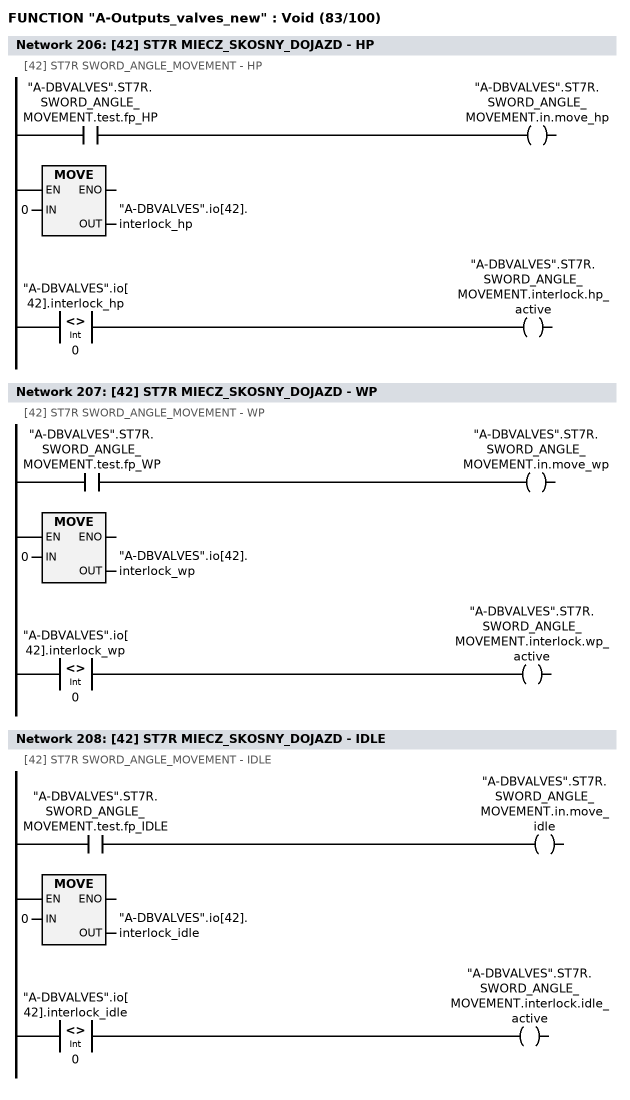
      O "A-DBVALVES".ST7R.SWORD_ANGLE_MOVEMENT.test.fp_HP;
//    O     "A-Flags".STATION.IN_HP_STEP
      = "A-DBVALVES".ST7R.SWORD_ANGLE_MOVEMENT.in.move_hp;

// Interlock hp
      L 0;
      T "A-DBVALVES".io[42].interlock_hp;

//{INTERLOCK_HP42}

      A(;
      L "A-DBVALVES".io[42].interlock_hp;
      L 0;
      <>I;
      );
      = "A-DBVALVES".ST7R.SWORD_ANGLE_MOVEMENT.interlock.hp_active;
NETWORK
TITLE = [42] ST7R MIECZ_SKOSNY_DOJAZD - WP
//[42] ST7R SWORD_ANGLE_MOVEMENT - WP
      O "A-DBVALVES".ST7R.SWORD_ANGLE_MOVEMENT.test.fp_WP;
      = "A-DBVALVES".ST7R.SWORD_ANGLE_MOVEMENT.in.move_wp;

// Interlock wp
      L 0;
      T "A-DBVALVES".io[42].interlock_wp;

//{INTERLOCK_WP42}

      A(;
      L "A-DBVALVES".io[42].interlock_wp;
      L 0;
      <>I;
      );
      = "A-DBVALVES".ST7R.SWORD_ANGLE_MOVEMENT.interlock.wp_active;
NETWORK
TITLE = [42] ST7R MIECZ_SKOSNY_DOJAZD - IDLE
//[42] ST7R SWORD_ANGLE_MOVEMENT - IDLE
      O "A-DBVALVES".ST7R.SWORD_ANGLE_MOVEMENT.test.fp_IDLE;
      = "A-DBVALVES".ST7R.SWORD_ANGLE_MOVEMENT.in.move_idle;

// Interlock idle
      L 0;
      T "A-DBVALVES".io[42].interlock_idle;

//{INTERLOCK_IDLE42}

      A(;
      L "A-DBVALVES".io[42].interlock_idle;
      L 0;
      <>I;
      );
      = "A-DBVALVES".ST7R.SWORD_ANGLE_MOVEMENT.interlock.idle_active;
NETWORK
TITLE = [42] ST7R MIECZ_SKOSNY_DOJAZD
//[42] ST7R SWORD_ANGLE_MOVEMENT
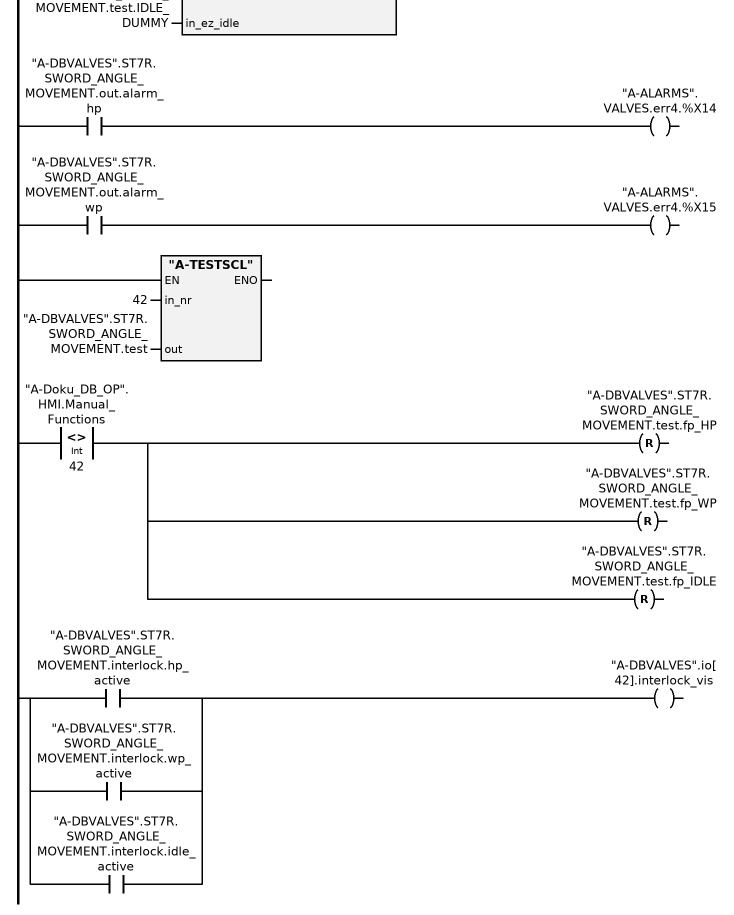
      CALL "3STATE_PISTON_with_brake", "INST_ST7R MIECZ_SKOSNY_DOJAZD"
      (  in_safety_on                := "A-Flags".STATION.SAFETY_OK ,
         in_curtain_on               := "A-Flags".STATION.CURTAIN.OK ,
         in_move_hp                  := "A-DBVALVES".ST7R.SWORD_ANGLE_MOVEMENT.in.move_hp ,
         in_move_wp                  := "A-DBVALVES".ST7R.SWORD_ANGLE_MOVEMENT.in.move_wp ,
         in_move_idle                := "A-DBVALVES".ST7R.SWORD_ANGLE_MOVEMENT.in.move_idle ,
         in_interlock_hp             := "A-DBVALVES".ST7R.SWORD_ANGLE_MOVEMENT.interlock.hp_active ,
         in_interlock_wp             := "A-DBVALVES".ST7R.SWORD_ANGLE_MOVEMENT.interlock.wp_active ,
         in_interlock_idle           := "A-DBVALVES".ST7R.SWORD_ANGLE_MOVEMENT.interlock.idle_active ,
         in_sensor_hp1               := "ST7R-vsen_sword_angle_movement_HP_right" ,
         in_sensor_hp2               := "ST7R-vsen_sword_angle_movement_HP_right" ,
         in_sensor_wp1               := "ST7R-vsen_sword_angle_movement_WP_front" ,
         in_sensor_wp2               := "ST7R-vsen_sword_angle_movement_WP_front" ,
         out_in_hp                   := "A-DBVALVES".ST7R.SWORD_ANGLE_MOVEMENT.out.in_hp ,
         out_in_wp                   := "A-DBVALVES".ST7R.SWORD_ANGLE_MOVEMENT.out.in_wp ,
         out_idle                    := "A-DBVALVES".ST7R.SWORD_ANGLE_MOVEMENT.out.in_idle ,
         out_status                  := "A-DBVALVES".ST7R.SWORD_ANGLE_MOVEMENT.out.status ,
         out_brake                   := #brake ,
         out_alarm_hp                := "A-DBVALVES".ST7R.SWORD_ANGLE_MOVEMENT.out.alarm_hp ,
         out_alarm_wp                := "A-DBVALVES".ST7R.SWORD_ANGLE_MOVEMENT.out.alarm_wp ,
         out_alarm_idle              := "A-DBVALVES".ST7R.SWORD_ANGLE_MOVEMENT.out.alarm_idle ,
         out_diag_status             := "A-DBVALVES".ST7R.SWORD_ANGLE_MOVEMENT.out.diag_status ,
         out_interlock_show          := "A-DBVALVES".ST7R.SWORD_ANGLE_MOVEMENT.interlock.active ,
         in_ez_hp                    := "ST7R-ez_sword_angle_movement_HP_right" ,
         in_ez_wp                    := "ST7R-ez_sword_angle_movement_WP_front" ,
         in_ez_idle                  := "A-DBVALVES".ST7R.SWORD_ANGLE_MOVEMENT.test.IDLE_DUMMY
      );

      CALL "3STATE_DIAG"
      (  in_diag_status              := "A-DBVALVES".ST7R.SWORD_ANGLE_MOVEMENT.out.diag_status ,
         in_Ipw1                     := 'I140.2' ,
         in_Ipw2                     := ' ' ,
         in_Ipr1                     := 'I141.2' ,
         in_Ipr2                     := ' ' ,
         in_Qpw                      := 'Q140.7' ,
         in_Qpr                      := 'Q141.7' ,
         in_tio                      := "A-DBVALVES".io[42]
      );

      A "A-DBVALVES".ST7R.SWORD_ANGLE_MOVEMENT.out.alarm_hp;
      = "A-ALARMS".VALVES.err4.%X14;

      A "A-DBVALVES".ST7R.SWORD_ANGLE_MOVEMENT.out.alarm_wp;
      = "A-ALARMS".VALVES.err4.%X15;

      CALL "A-TESTSCL"
      (  in_nr                       := 42 ,
         out                         := "A-DBVALVES".ST7R.SWORD_ANGLE_MOVEMENT.test
      );

      A(;
      L "A-Doku_DB_OP".HMI.Manual_Functions;
      L 42;
      <>I;
      );
      R "A-DBVALVES".ST7R.SWORD_ANGLE_MOVEMENT.test.fp_HP;
      R "A-DBVALVES".ST7R.SWORD_ANGLE_MOVEMENT.test.fp_WP;
      R "A-DBVALVES".ST7R.SWORD_ANGLE_MOVEMENT.test.fp_IDLE;

      O "A-DBVALVES".ST7R.SWORD_ANGLE_MOVEMENT.interlock.hp_active;
      O "A-DBVALVES".ST7R.SWORD_ANGLE_MOVEMENT.interlock.wp_active;
      O "A-DBVALVES".ST7R.SWORD_ANGLE_MOVEMENT.interlock.idle_active;
      = "A-DBVALVES".io[42].interlock_vis;
NETWORK
TITLE = -

NETWORK
TITLE = [43] ST7R MIECZ_PROSTY_DOJAZD - HP
//[43] ST7R SWORD_STRAIGHT_MOVEMENT - HP
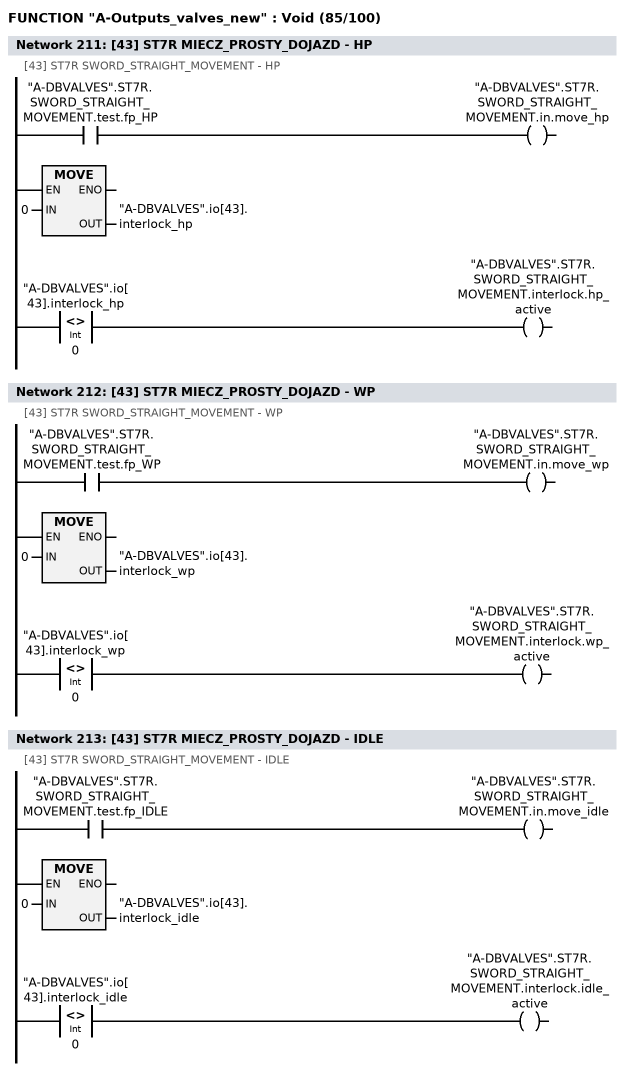
      O "A-DBVALVES".ST7R.SWORD_STRAIGHT_MOVEMENT.test.fp_HP;
//    O     "A-Flags".STATION.IN_HP_STEP
      = "A-DBVALVES".ST7R.SWORD_STRAIGHT_MOVEMENT.in.move_hp;

// Interlock hp
      L 0;
      T "A-DBVALVES".io[43].interlock_hp;

//{INTERLOCK_HP43}

      A(;
      L "A-DBVALVES".io[43].interlock_hp;
      L 0;
      <>I;
      );
      = "A-DBVALVES".ST7R.SWORD_STRAIGHT_MOVEMENT.interlock.hp_active;
NETWORK
TITLE = [43] ST7R MIECZ_PROSTY_DOJAZD - WP
//[43] ST7R SWORD_STRAIGHT_MOVEMENT - WP
      O "A-DBVALVES".ST7R.SWORD_STRAIGHT_MOVEMENT.test.fp_WP;
      = "A-DBVALVES".ST7R.SWORD_STRAIGHT_MOVEMENT.in.move_wp;

// Interlock wp
      L 0;
      T "A-DBVALVES".io[43].interlock_wp;

//{INTERLOCK_WP43}

      A(;
      L "A-DBVALVES".io[43].interlock_wp;
      L 0;
      <>I;
      );
      = "A-DBVALVES".ST7R.SWORD_STRAIGHT_MOVEMENT.interlock.wp_active;
NETWORK
TITLE = [43] ST7R MIECZ_PROSTY_DOJAZD - IDLE
//[43] ST7R SWORD_STRAIGHT_MOVEMENT - IDLE
      O "A-DBVALVES".ST7R.SWORD_STRAIGHT_MOVEMENT.test.fp_IDLE;
      = "A-DBVALVES".ST7R.SWORD_STRAIGHT_MOVEMENT.in.move_idle;

// Interlock idle
      L 0;
      T "A-DBVALVES".io[43].interlock_idle;

//{INTERLOCK_IDLE43}

      A(;
      L "A-DBVALVES".io[43].interlock_idle;
      L 0;
      <>I;
      );
      = "A-DBVALVES".ST7R.SWORD_STRAIGHT_MOVEMENT.interlock.idle_active;
NETWORK
TITLE = [43] ST7R MIECZ_PROSTY_DOJAZD
//[43] ST7R SWORD_STRAIGHT_MOVEMENT
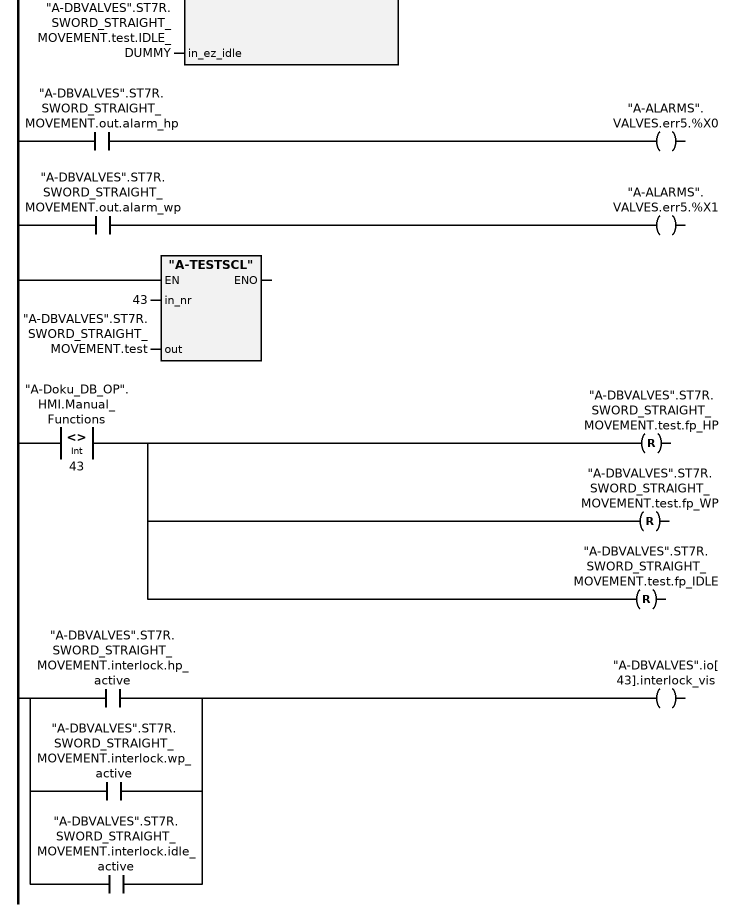
      CALL "3STATE_PISTON_with_brake", "INST_ST7R MIECZ_PROSTY_DOJAZD"
      (  in_safety_on                := "A-Flags".STATION.SAFETY_OK ,
         in_curtain_on               := "A-Flags".STATION.CURTAIN.OK ,
         in_move_hp                  := "A-DBVALVES".ST7R.SWORD_STRAIGHT_MOVEMENT.in.move_hp ,
         in_move_wp                  := "A-DBVALVES".ST7R.SWORD_STRAIGHT_MOVEMENT.in.move_wp ,
         in_move_idle                := "A-DBVALVES".ST7R.SWORD_STRAIGHT_MOVEMENT.in.move_idle ,
         in_interlock_hp             := "A-DBVALVES".ST7R.SWORD_STRAIGHT_MOVEMENT.interlock.hp_active ,
         in_interlock_wp             := "A-DBVALVES".ST7R.SWORD_STRAIGHT_MOVEMENT.interlock.wp_active ,
         in_interlock_idle           := "A-DBVALVES".ST7R.SWORD_STRAIGHT_MOVEMENT.interlock.idle_active ,
         in_sensor_hp1               := "ST7R-vsen_sword_straight_movement_HP_right" ,
         in_sensor_hp2               := "ST7R-vsen_sword_straight_movement_HP_right" ,
         in_sensor_wp1               := "ST7R-vsen_sword_straight_movement_WP_front" ,
         in_sensor_wp2               := "ST7R-vsen_sword_straight_movement_WP_front" ,
         out_in_hp                   := "A-DBVALVES".ST7R.SWORD_STRAIGHT_MOVEMENT.out.in_hp ,
         out_in_wp                   := "A-DBVALVES".ST7R.SWORD_STRAIGHT_MOVEMENT.out.in_wp ,
         out_idle                    := "A-DBVALVES".ST7R.SWORD_STRAIGHT_MOVEMENT.out.in_idle ,
         out_status                  := "A-DBVALVES".ST7R.SWORD_STRAIGHT_MOVEMENT.out.status ,
         out_brake                   := #brake ,
         out_alarm_hp                := "A-DBVALVES".ST7R.SWORD_STRAIGHT_MOVEMENT.out.alarm_hp ,
         out_alarm_wp                := "A-DBVALVES".ST7R.SWORD_STRAIGHT_MOVEMENT.out.alarm_wp ,
         out_alarm_idle              := "A-DBVALVES".ST7R.SWORD_STRAIGHT_MOVEMENT.out.alarm_idle ,
         out_diag_status             := "A-DBVALVES".ST7R.SWORD_STRAIGHT_MOVEMENT.out.diag_status ,
         out_interlock_show          := "A-DBVALVES".ST7R.SWORD_STRAIGHT_MOVEMENT.interlock.active ,
         in_ez_hp                    := "ST7R-ez_sword_straight_movement_HP_right" ,
         in_ez_wp                    := "ST7R-ez_sword_straight_movement_WP_front" ,
         in_ez_idle                  := "A-DBVALVES".ST7R.SWORD_STRAIGHT_MOVEMENT.test.IDLE_DUMMY
      );

      CALL "3STATE_DIAG"
      (  in_diag_status              := "A-DBVALVES".ST7R.SWORD_STRAIGHT_MOVEMENT.out.diag_status ,
         in_Ipw1                     := 'I130.0' ,
         in_Ipw2                     := ' ' ,
         in_Ipr1                     := 'I131.0' ,
         in_Ipr2                     := ' ' ,
         in_Qpw                      := 'Q3012.1' ,
         in_Qpr                      := 'Q3012.0' ,
         in_tio                      := "A-DBVALVES".io[43]
      );

      A "A-DBVALVES".ST7R.SWORD_STRAIGHT_MOVEMENT.out.alarm_hp;
      = "A-ALARMS".VALVES.err5.%X0;

      A "A-DBVALVES".ST7R.SWORD_STRAIGHT_MOVEMENT.out.alarm_wp;
      = "A-ALARMS".VALVES.err5.%X1;

      CALL "A-TESTSCL"
      (  in_nr                       := 43 ,
         out                         := "A-DBVALVES".ST7R.SWORD_STRAIGHT_MOVEMENT.test
      );

      A(;
      L "A-Doku_DB_OP".HMI.Manual_Functions;
      L 43;
      <>I;
      );
      R "A-DBVALVES".ST7R.SWORD_STRAIGHT_MOVEMENT.test.fp_HP;
      R "A-DBVALVES".ST7R.SWORD_STRAIGHT_MOVEMENT.test.fp_WP;
      R "A-DBVALVES".ST7R.SWORD_STRAIGHT_MOVEMENT.test.fp_IDLE;

      O "A-DBVALVES".ST7R.SWORD_STRAIGHT_MOVEMENT.interlock.hp_active;
      O "A-DBVALVES".ST7R.SWORD_STRAIGHT_MOVEMENT.interlock.wp_active;
      O "A-DBVALVES".ST7R.SWORD_STRAIGHT_MOVEMENT.interlock.idle_active;
      = "A-DBVALVES".io[43].interlock_vis;
NETWORK
TITLE = -

NETWORK
TITLE = [44] ST7R MIECZ_PROSTY - HP
//[44] ST7R SWORD_STRAIGHT - HP
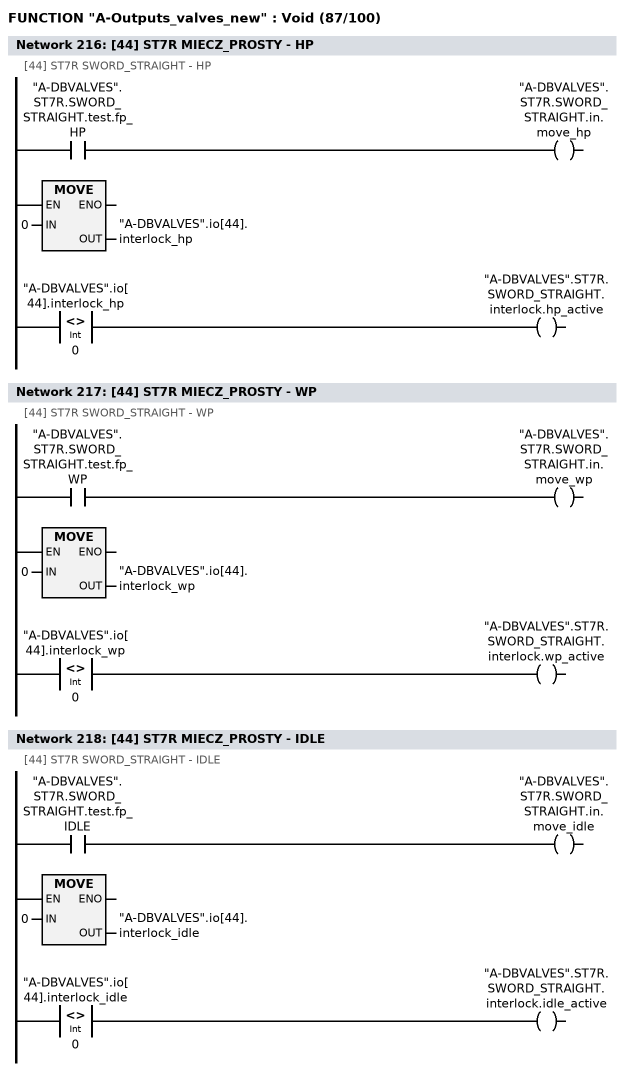
      O "A-DBVALVES".ST7R.SWORD_STRAIGHT.test.fp_HP;
//    O     "A-Flags".STATION.IN_HP_STEP
      = "A-DBVALVES".ST7R.SWORD_STRAIGHT.in.move_hp;

// Interlock hp
      L 0;
      T "A-DBVALVES".io[44].interlock_hp;

//{INTERLOCK_HP44}

      A(;
      L "A-DBVALVES".io[44].interlock_hp;
      L 0;
      <>I;
      );
      = "A-DBVALVES".ST7R.SWORD_STRAIGHT.interlock.hp_active;
NETWORK
TITLE = [44] ST7R MIECZ_PROSTY - WP
//[44] ST7R SWORD_STRAIGHT - WP
      O "A-DBVALVES".ST7R.SWORD_STRAIGHT.test.fp_WP;
      = "A-DBVALVES".ST7R.SWORD_STRAIGHT.in.move_wp;

// Interlock wp
      L 0;
      T "A-DBVALVES".io[44].interlock_wp;

//{INTERLOCK_WP44}

      A(;
      L "A-DBVALVES".io[44].interlock_wp;
      L 0;
      <>I;
      );
      = "A-DBVALVES".ST7R.SWORD_STRAIGHT.interlock.wp_active;
NETWORK
TITLE = [44] ST7R MIECZ_PROSTY - IDLE
//[44] ST7R SWORD_STRAIGHT - IDLE
      O "A-DBVALVES".ST7R.SWORD_STRAIGHT.test.fp_IDLE;
      = "A-DBVALVES".ST7R.SWORD_STRAIGHT.in.move_idle;

// Interlock idle
      L 0;
      T "A-DBVALVES".io[44].interlock_idle;

//{INTERLOCK_IDLE44}

      A(;
      L "A-DBVALVES".io[44].interlock_idle;
      L 0;
      <>I;
      );
      = "A-DBVALVES".ST7R.SWORD_STRAIGHT.interlock.idle_active;
NETWORK
TITLE = [44] ST7R MIECZ_PROSTY
//[44] ST7R SWORD_STRAIGHT
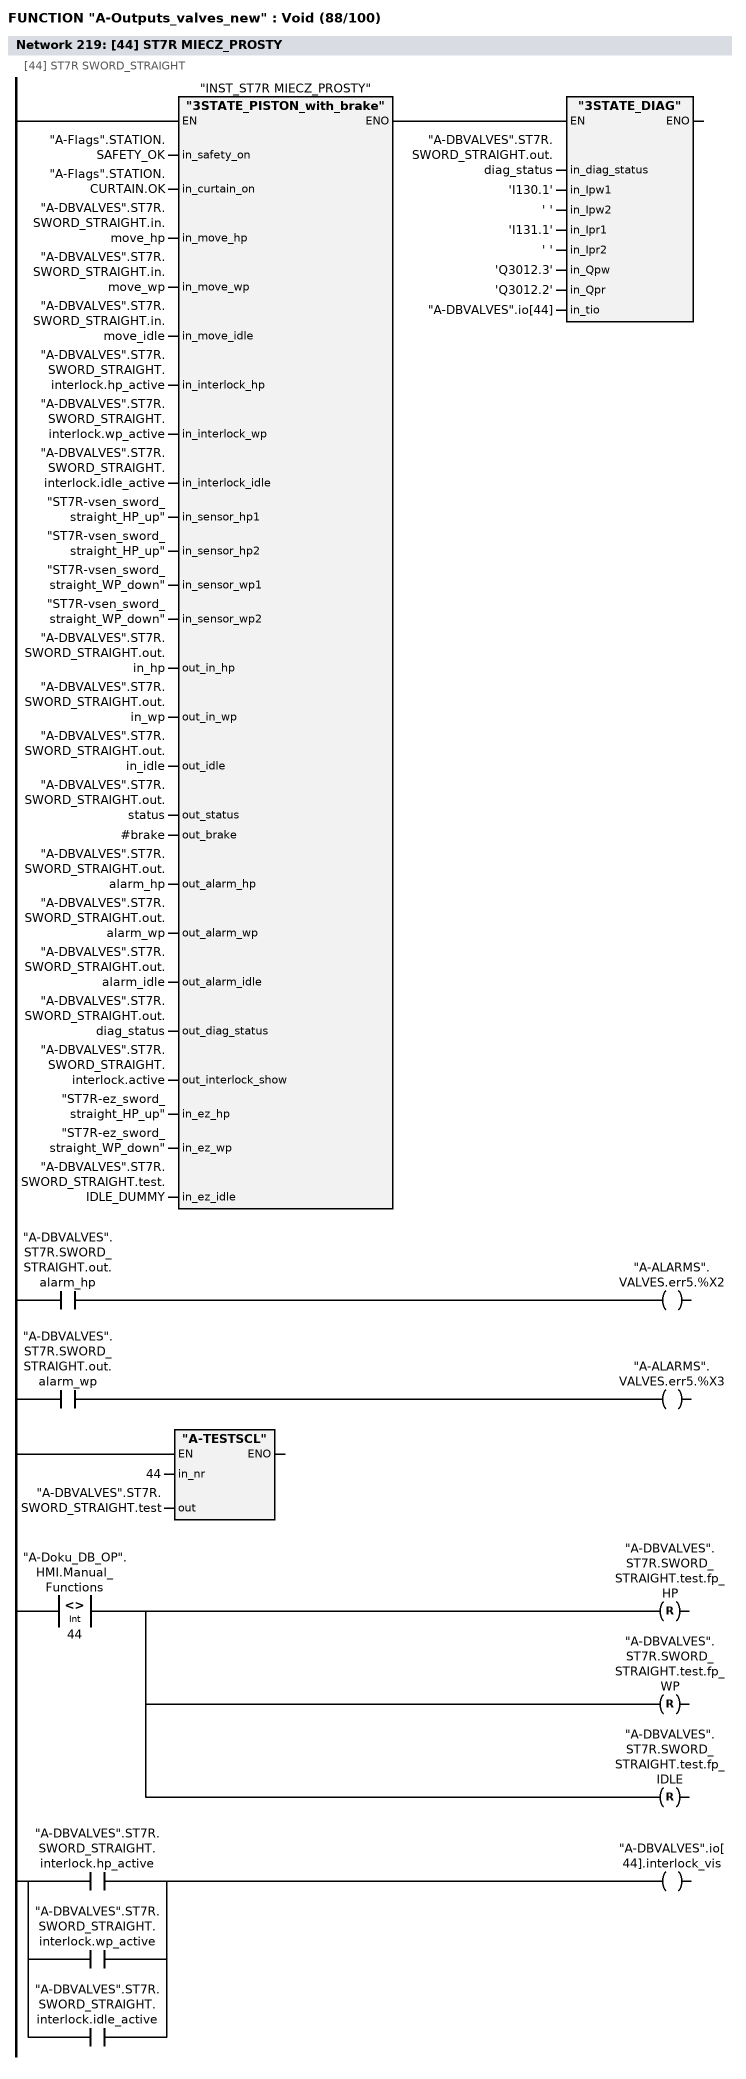
      CALL "3STATE_PISTON_with_brake", "INST_ST7R MIECZ_PROSTY"
      (  in_safety_on                := "A-Flags".STATION.SAFETY_OK ,
         in_curtain_on               := "A-Flags".STATION.CURTAIN.OK ,
         in_move_hp                  := "A-DBVALVES".ST7R.SWORD_STRAIGHT.in.move_hp ,
         in_move_wp                  := "A-DBVALVES".ST7R.SWORD_STRAIGHT.in.move_wp ,
         in_move_idle                := "A-DBVALVES".ST7R.SWORD_STRAIGHT.in.move_idle ,
         in_interlock_hp             := "A-DBVALVES".ST7R.SWORD_STRAIGHT.interlock.hp_active ,
         in_interlock_wp             := "A-DBVALVES".ST7R.SWORD_STRAIGHT.interlock.wp_active ,
         in_interlock_idle           := "A-DBVALVES".ST7R.SWORD_STRAIGHT.interlock.idle_active ,
         in_sensor_hp1               := "ST7R-vsen_sword_straight_HP_up" ,
         in_sensor_hp2               := "ST7R-vsen_sword_straight_HP_up" ,
         in_sensor_wp1               := "ST7R-vsen_sword_straight_WP_down" ,
         in_sensor_wp2               := "ST7R-vsen_sword_straight_WP_down" ,
         out_in_hp                   := "A-DBVALVES".ST7R.SWORD_STRAIGHT.out.in_hp ,
         out_in_wp                   := "A-DBVALVES".ST7R.SWORD_STRAIGHT.out.in_wp ,
         out_idle                    := "A-DBVALVES".ST7R.SWORD_STRAIGHT.out.in_idle ,
         out_status                  := "A-DBVALVES".ST7R.SWORD_STRAIGHT.out.status ,
         out_brake                   := #brake ,
         out_alarm_hp                := "A-DBVALVES".ST7R.SWORD_STRAIGHT.out.alarm_hp ,
         out_alarm_wp                := "A-DBVALVES".ST7R.SWORD_STRAIGHT.out.alarm_wp ,
         out_alarm_idle              := "A-DBVALVES".ST7R.SWORD_STRAIGHT.out.alarm_idle ,
         out_diag_status             := "A-DBVALVES".ST7R.SWORD_STRAIGHT.out.diag_status ,
         out_interlock_show          := "A-DBVALVES".ST7R.SWORD_STRAIGHT.interlock.active ,
         in_ez_hp                    := "ST7R-ez_sword_straight_HP_up" ,
         in_ez_wp                    := "ST7R-ez_sword_straight_WP_down" ,
         in_ez_idle                  := "A-DBVALVES".ST7R.SWORD_STRAIGHT.test.IDLE_DUMMY
      );

      CALL "3STATE_DIAG"
      (  in_diag_status              := "A-DBVALVES".ST7R.SWORD_STRAIGHT.out.diag_status ,
         in_Ipw1                     := 'I130.1' ,
         in_Ipw2                     := ' ' ,
         in_Ipr1                     := 'I131.1' ,
         in_Ipr2                     := ' ' ,
         in_Qpw                      := 'Q3012.3' ,
         in_Qpr                      := 'Q3012.2' ,
         in_tio                      := "A-DBVALVES".io[44]
      );

      A "A-DBVALVES".ST7R.SWORD_STRAIGHT.out.alarm_hp;
      = "A-ALARMS".VALVES.err5.%X2;

      A "A-DBVALVES".ST7R.SWORD_STRAIGHT.out.alarm_wp;
      = "A-ALARMS".VALVES.err5.%X3;

      CALL "A-TESTSCL"
      (  in_nr                       := 44 ,
         out                         := "A-DBVALVES".ST7R.SWORD_STRAIGHT.test
      );

      A(;
      L "A-Doku_DB_OP".HMI.Manual_Functions;
      L 44;
      <>I;
      );
      R "A-DBVALVES".ST7R.SWORD_STRAIGHT.test.fp_HP;
      R "A-DBVALVES".ST7R.SWORD_STRAIGHT.test.fp_WP;
      R "A-DBVALVES".ST7R.SWORD_STRAIGHT.test.fp_IDLE;

      O "A-DBVALVES".ST7R.SWORD_STRAIGHT.interlock.hp_active;
      O "A-DBVALVES".ST7R.SWORD_STRAIGHT.interlock.wp_active;
      O "A-DBVALVES".ST7R.SWORD_STRAIGHT.interlock.idle_active;
      = "A-DBVALVES".io[44].interlock_vis;
NETWORK
TITLE = -

NETWORK
TITLE = [45] ST7R MIECZ_RUCHOMY_DOJAZD - HP
//[45] ST7R SWORD_MOBILE_MOVEMENT - HP
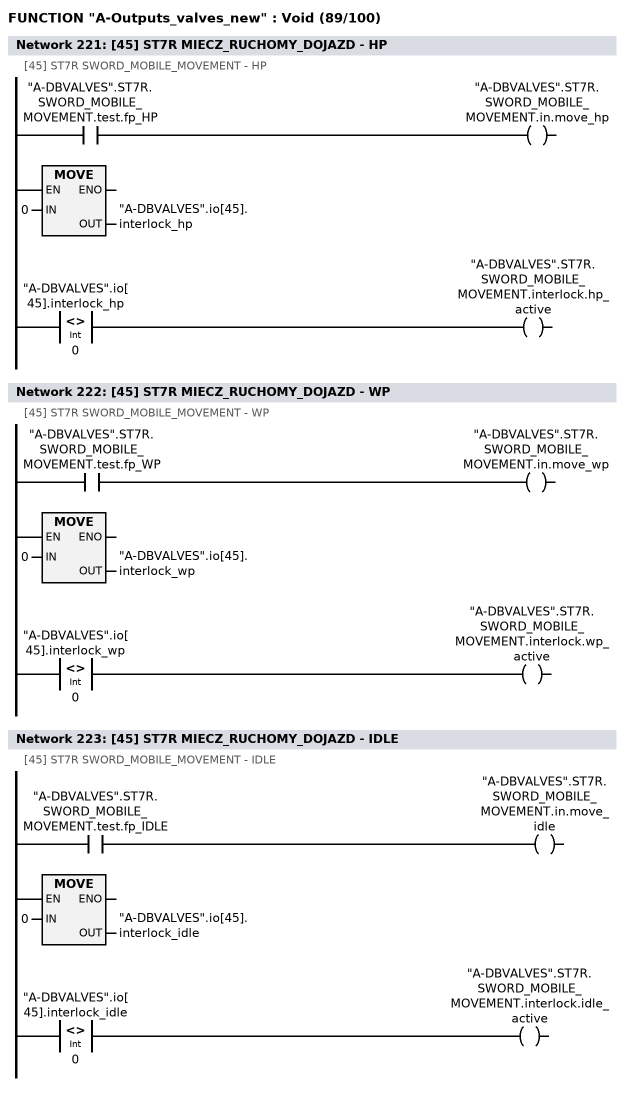
      O "A-DBVALVES".ST7R.SWORD_MOBILE_MOVEMENT.test.fp_HP;
//    O     "A-Flags".STATION.IN_HP_STEP
      = "A-DBVALVES".ST7R.SWORD_MOBILE_MOVEMENT.in.move_hp;

// Interlock hp
      L 0;
      T "A-DBVALVES".io[45].interlock_hp;

//{INTERLOCK_HP45}

      A(;
      L "A-DBVALVES".io[45].interlock_hp;
      L 0;
      <>I;
      );
      = "A-DBVALVES".ST7R.SWORD_MOBILE_MOVEMENT.interlock.hp_active;
NETWORK
TITLE = [45] ST7R MIECZ_RUCHOMY_DOJAZD - WP
//[45] ST7R SWORD_MOBILE_MOVEMENT - WP
      O "A-DBVALVES".ST7R.SWORD_MOBILE_MOVEMENT.test.fp_WP;
      = "A-DBVALVES".ST7R.SWORD_MOBILE_MOVEMENT.in.move_wp;

// Interlock wp
      L 0;
      T "A-DBVALVES".io[45].interlock_wp;

//{INTERLOCK_WP45}

      A(;
      L "A-DBVALVES".io[45].interlock_wp;
      L 0;
      <>I;
      );
      = "A-DBVALVES".ST7R.SWORD_MOBILE_MOVEMENT.interlock.wp_active;
NETWORK
TITLE = [45] ST7R MIECZ_RUCHOMY_DOJAZD - IDLE
//[45] ST7R SWORD_MOBILE_MOVEMENT - IDLE
      O "A-DBVALVES".ST7R.SWORD_MOBILE_MOVEMENT.test.fp_IDLE;
      = "A-DBVALVES".ST7R.SWORD_MOBILE_MOVEMENT.in.move_idle;

// Interlock idle
      L 0;
      T "A-DBVALVES".io[45].interlock_idle;

//{INTERLOCK_IDLE45}

      A(;
      L "A-DBVALVES".io[45].interlock_idle;
      L 0;
      <>I;
      );
      = "A-DBVALVES".ST7R.SWORD_MOBILE_MOVEMENT.interlock.idle_active;
NETWORK
TITLE = [45] ST7R MIECZ_RUCHOMY_DOJAZD
//[45] ST7R SWORD_MOBILE_MOVEMENT
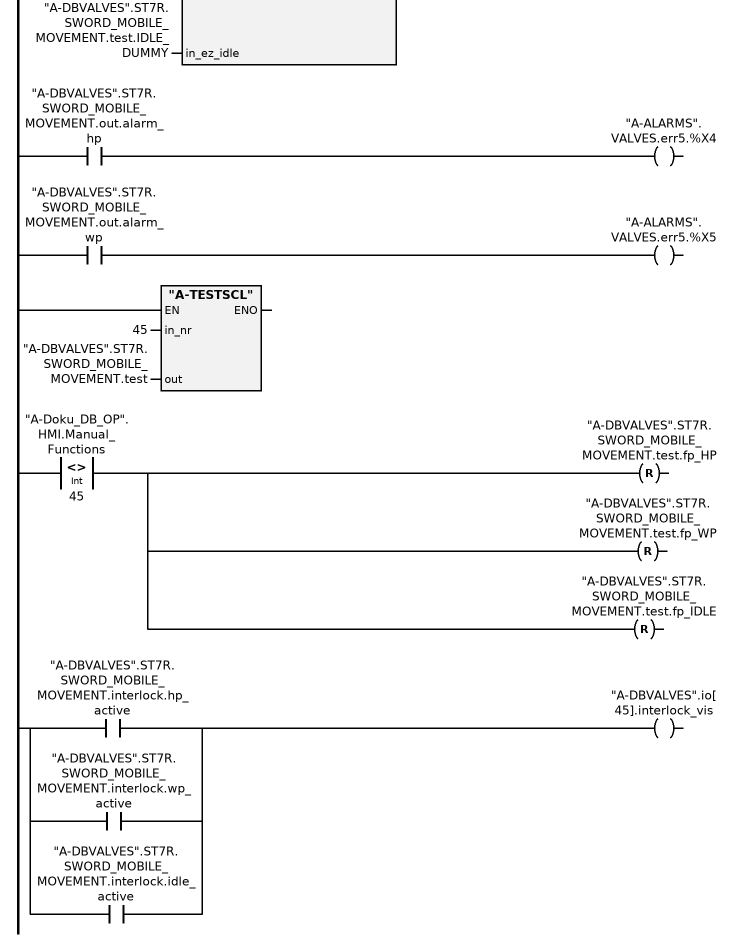
      CALL "3STATE_PISTON_with_brake", "INST_ST7R MIECZ_RUCHOMY_DOJAZD"
      (  in_safety_on                := "A-Flags".STATION.SAFETY_OK ,
         in_curtain_on               := "A-Flags".STATION.CURTAIN.OK ,
         in_move_hp                  := "A-DBVALVES".ST7R.SWORD_MOBILE_MOVEMENT.in.move_hp ,
         in_move_wp                  := "A-DBVALVES".ST7R.SWORD_MOBILE_MOVEMENT.in.move_wp ,
         in_move_idle                := "A-DBVALVES".ST7R.SWORD_MOBILE_MOVEMENT.in.move_idle ,
         in_interlock_hp             := "A-DBVALVES".ST7R.SWORD_MOBILE_MOVEMENT.interlock.hp_active ,
         in_interlock_wp             := "A-DBVALVES".ST7R.SWORD_MOBILE_MOVEMENT.interlock.wp_active ,
         in_interlock_idle           := "A-DBVALVES".ST7R.SWORD_MOBILE_MOVEMENT.interlock.idle_active ,
         in_sensor_hp1               := "ST7R-vsen_sword_mobile_movement_HP_right" ,
         in_sensor_hp2               := "ST7R-vsen_sword_mobile_movement_HP_right" ,
         in_sensor_wp1               := "ST7R-vsen_sword_mobile_movement_WP_front" ,
         in_sensor_wp2               := "ST7R-vsen_sword_mobile_movement_WP_front" ,
         out_in_hp                   := "A-DBVALVES".ST7R.SWORD_MOBILE_MOVEMENT.out.in_hp ,
         out_in_wp                   := "A-DBVALVES".ST7R.SWORD_MOBILE_MOVEMENT.out.in_wp ,
         out_idle                    := "A-DBVALVES".ST7R.SWORD_MOBILE_MOVEMENT.out.in_idle ,
         out_status                  := "A-DBVALVES".ST7R.SWORD_MOBILE_MOVEMENT.out.status ,
         out_brake                   := #brake ,
         out_alarm_hp                := "A-DBVALVES".ST7R.SWORD_MOBILE_MOVEMENT.out.alarm_hp ,
         out_alarm_wp                := "A-DBVALVES".ST7R.SWORD_MOBILE_MOVEMENT.out.alarm_wp ,
         out_alarm_idle              := "A-DBVALVES".ST7R.SWORD_MOBILE_MOVEMENT.out.alarm_idle ,
         out_diag_status             := "A-DBVALVES".ST7R.SWORD_MOBILE_MOVEMENT.out.diag_status ,
         out_interlock_show          := "A-DBVALVES".ST7R.SWORD_MOBILE_MOVEMENT.interlock.active ,
         in_ez_hp                    := "ST7R-ez_sword_mobile_movement_HP_right" ,
         in_ez_wp                    := "ST7R-ez_sword_mobile_movement_WP_front" ,
         in_ez_idle                  := "A-DBVALVES".ST7R.SWORD_MOBILE_MOVEMENT.test.IDLE_DUMMY
      );

      CALL "3STATE_DIAG"
      (  in_diag_status              := "A-DBVALVES".ST7R.SWORD_MOBILE_MOVEMENT.out.diag_status ,
         in_Ipw1                     := 'I130.3' ,
         in_Ipw2                     := ' ' ,
         in_Ipr1                     := 'I131.3' ,
         in_Ipr2                     := ' ' ,
         in_Qpw                      := 'Q3012.7' ,
         in_Qpr                      := 'Q3012.6' ,
         in_tio                      := "A-DBVALVES".io[45]
      );

      A "A-DBVALVES".ST7R.SWORD_MOBILE_MOVEMENT.out.alarm_hp;
      = "A-ALARMS".VALVES.err5.%X4;

      A "A-DBVALVES".ST7R.SWORD_MOBILE_MOVEMENT.out.alarm_wp;
      = "A-ALARMS".VALVES.err5.%X5;

      CALL "A-TESTSCL"
      (  in_nr                       := 45 ,
         out                         := "A-DBVALVES".ST7R.SWORD_MOBILE_MOVEMENT.test
      );

      A(;
      L "A-Doku_DB_OP".HMI.Manual_Functions;
      L 45;
      <>I;
      );
      R "A-DBVALVES".ST7R.SWORD_MOBILE_MOVEMENT.test.fp_HP;
      R "A-DBVALVES".ST7R.SWORD_MOBILE_MOVEMENT.test.fp_WP;
      R "A-DBVALVES".ST7R.SWORD_MOBILE_MOVEMENT.test.fp_IDLE;

      O "A-DBVALVES".ST7R.SWORD_MOBILE_MOVEMENT.interlock.hp_active;
      O "A-DBVALVES".ST7R.SWORD_MOBILE_MOVEMENT.interlock.wp_active;
      O "A-DBVALVES".ST7R.SWORD_MOBILE_MOVEMENT.interlock.idle_active;
      = "A-DBVALVES".io[45].interlock_vis;
NETWORK
TITLE = -

NETWORK
TITLE = [46] ST7R MIECZ_RUCHOMY_PRZEJAZD - HP
//[46] ST7R SWORD_MOBILE_SLIDE - HP
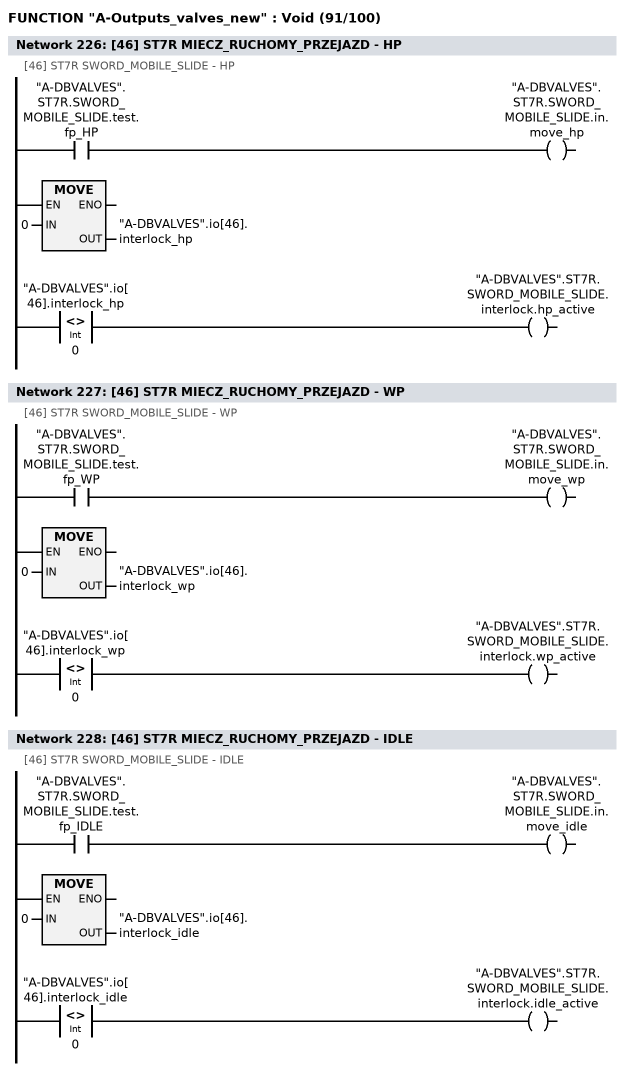
      O "A-DBVALVES".ST7R.SWORD_MOBILE_SLIDE.test.fp_HP;
//    O     "A-Flags".STATION.IN_HP_STEP
      = "A-DBVALVES".ST7R.SWORD_MOBILE_SLIDE.in.move_hp;

// Interlock hp
      L 0;
      T "A-DBVALVES".io[46].interlock_hp;

//{INTERLOCK_HP46}

      A(;
      L "A-DBVALVES".io[46].interlock_hp;
      L 0;
      <>I;
      );
      = "A-DBVALVES".ST7R.SWORD_MOBILE_SLIDE.interlock.hp_active;
NETWORK
TITLE = [46] ST7R MIECZ_RUCHOMY_PRZEJAZD - WP
//[46] ST7R SWORD_MOBILE_SLIDE - WP
      O "A-DBVALVES".ST7R.SWORD_MOBILE_SLIDE.test.fp_WP;
      = "A-DBVALVES".ST7R.SWORD_MOBILE_SLIDE.in.move_wp;

// Interlock wp
      L 0;
      T "A-DBVALVES".io[46].interlock_wp;

//{INTERLOCK_WP46}

      A(;
      L "A-DBVALVES".io[46].interlock_wp;
      L 0;
      <>I;
      );
      = "A-DBVALVES".ST7R.SWORD_MOBILE_SLIDE.interlock.wp_active;
NETWORK
TITLE = [46] ST7R MIECZ_RUCHOMY_PRZEJAZD - IDLE
//[46] ST7R SWORD_MOBILE_SLIDE - IDLE
      O "A-DBVALVES".ST7R.SWORD_MOBILE_SLIDE.test.fp_IDLE;
      = "A-DBVALVES".ST7R.SWORD_MOBILE_SLIDE.in.move_idle;

// Interlock idle
      L 0;
      T "A-DBVALVES".io[46].interlock_idle;

//{INTERLOCK_IDLE46}

      A(;
      L "A-DBVALVES".io[46].interlock_idle;
      L 0;
      <>I;
      );
      = "A-DBVALVES".ST7R.SWORD_MOBILE_SLIDE.interlock.idle_active;
NETWORK
TITLE = [46] ST7R MIECZ_RUCHOMY_PRZEJAZD
//[46] ST7R SWORD_MOBILE_SLIDE
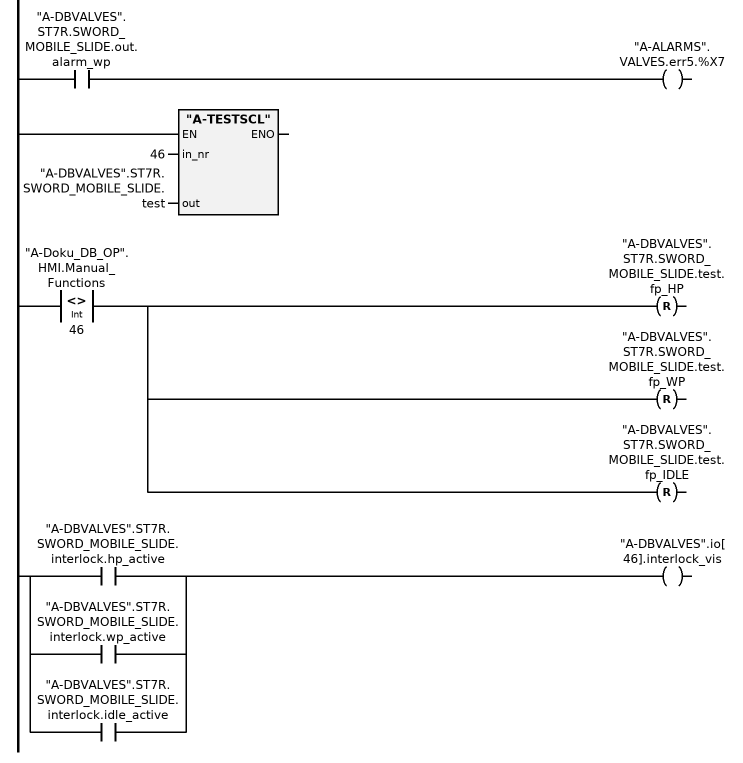
      CALL "3STATE_PISTON_with_brake", "INST_ST7R MIECZ_RUCHOMY_PRZEJAZD"
      (  in_safety_on                := "A-Flags".STATION.SAFETY_OK ,
         in_curtain_on               := "A-Flags".STATION.CURTAIN.OK ,
         in_move_hp                  := "A-DBVALVES".ST7R.SWORD_MOBILE_SLIDE.in.move_hp ,
         in_move_wp                  := "A-DBVALVES".ST7R.SWORD_MOBILE_SLIDE.in.move_wp ,
         in_move_idle                := "A-DBVALVES".ST7R.SWORD_MOBILE_SLIDE.in.move_idle ,
         in_interlock_hp             := "A-DBVALVES".ST7R.SWORD_MOBILE_SLIDE.interlock.hp_active ,
         in_interlock_wp             := "A-DBVALVES".ST7R.SWORD_MOBILE_SLIDE.interlock.wp_active ,
         in_interlock_idle           := "A-DBVALVES".ST7R.SWORD_MOBILE_SLIDE.interlock.idle_active ,
         in_sensor_hp1               := "ST7R-vsen_sword_mobile_slide_HP_right" ,
         in_sensor_hp2               := "ST7R-vsen_sword_mobile_slide_HP_right" ,
         in_sensor_wp1               := "ST7R-vsen_sword_mobile_slide_WP_left" ,
         in_sensor_wp2               := "ST7R-vsen_sword_mobile_slide_WP_left" ,
         out_in_hp                   := "A-DBVALVES".ST7R.SWORD_MOBILE_SLIDE.out.in_hp ,
         out_in_wp                   := "A-DBVALVES".ST7R.SWORD_MOBILE_SLIDE.out.in_wp ,
         out_idle                    := "A-DBVALVES".ST7R.SWORD_MOBILE_SLIDE.out.in_idle ,
         out_status                  := "A-DBVALVES".ST7R.SWORD_MOBILE_SLIDE.out.status ,
         out_brake                   := #brake ,
         out_alarm_hp                := "A-DBVALVES".ST7R.SWORD_MOBILE_SLIDE.out.alarm_hp ,
         out_alarm_wp                := "A-DBVALVES".ST7R.SWORD_MOBILE_SLIDE.out.alarm_wp ,
         out_alarm_idle              := "A-DBVALVES".ST7R.SWORD_MOBILE_SLIDE.out.alarm_idle ,
         out_diag_status             := "A-DBVALVES".ST7R.SWORD_MOBILE_SLIDE.out.diag_status ,
         out_interlock_show          := "A-DBVALVES".ST7R.SWORD_MOBILE_SLIDE.interlock.active ,
         in_ez_hp                    := "ST7R-ez_sword_mobile_slide_HP_right" ,
         in_ez_wp                    := "ST7R-ez_sword_mobile_slide_WP_left" ,
         in_ez_idle                  := "A-DBVALVES".ST7R.SWORD_MOBILE_SLIDE.test.IDLE_DUMMY
      );

      CALL "3STATE_DIAG"
      (  in_diag_status              := "A-DBVALVES".ST7R.SWORD_MOBILE_SLIDE.out.diag_status ,
         in_Ipw1                     := 'I130.2' ,
         in_Ipw2                     := ' ' ,
         in_Ipr1                     := 'I131.2' ,
         in_Ipr2                     := ' ' ,
         in_Qpw                      := 'Q3012.5' ,
         in_Qpr                      := 'Q3012.4' ,
         in_tio                      := "A-DBVALVES".io[46]
      );

      A "A-DBVALVES".ST7R.SWORD_MOBILE_SLIDE.out.alarm_hp;
      = "A-ALARMS".VALVES.err5.%X6;

      A "A-DBVALVES".ST7R.SWORD_MOBILE_SLIDE.out.alarm_wp;
      = "A-ALARMS".VALVES.err5.%X7;

      CALL "A-TESTSCL"
      (  in_nr                       := 46 ,
         out                         := "A-DBVALVES".ST7R.SWORD_MOBILE_SLIDE.test
      );

      A(;
      L "A-Doku_DB_OP".HMI.Manual_Functions;
      L 46;
      <>I;
      );
      R "A-DBVALVES".ST7R.SWORD_MOBILE_SLIDE.test.fp_HP;
      R "A-DBVALVES".ST7R.SWORD_MOBILE_SLIDE.test.fp_WP;
      R "A-DBVALVES".ST7R.SWORD_MOBILE_SLIDE.test.fp_IDLE;

      O "A-DBVALVES".ST7R.SWORD_MOBILE_SLIDE.interlock.hp_active;
      O "A-DBVALVES".ST7R.SWORD_MOBILE_SLIDE.interlock.wp_active;
      O "A-DBVALVES".ST7R.SWORD_MOBILE_SLIDE.interlock.idle_active;
      = "A-DBVALVES".io[46].interlock_vis;
NETWORK
TITLE = -

NETWORK
TITLE = [47] ST7R MIECZ_RUCHOMY - HP
//[47] ST7R SWORD_MOBILE - HP
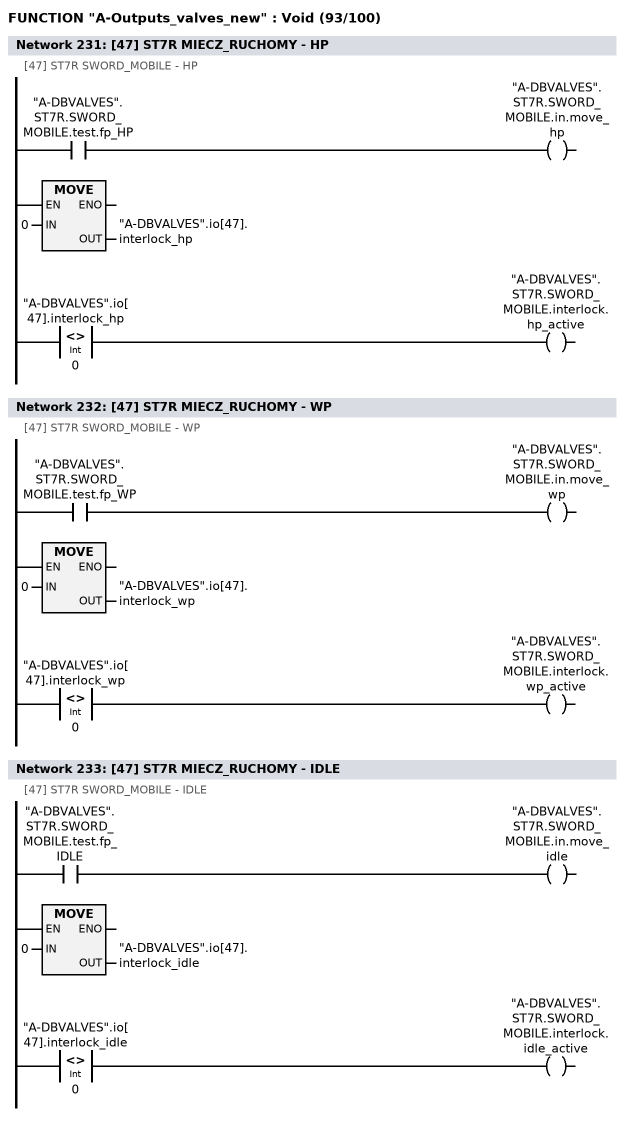
      O "A-DBVALVES".ST7R.SWORD_MOBILE.test.fp_HP;
//    O     "A-Flags".STATION.IN_HP_STEP
      = "A-DBVALVES".ST7R.SWORD_MOBILE.in.move_hp;

// Interlock hp
      L 0;
      T "A-DBVALVES".io[47].interlock_hp;

//{INTERLOCK_HP47}

      A(;
      L "A-DBVALVES".io[47].interlock_hp;
      L 0;
      <>I;
      );
      = "A-DBVALVES".ST7R.SWORD_MOBILE.interlock.hp_active;
NETWORK
TITLE = [47] ST7R MIECZ_RUCHOMY - WP
//[47] ST7R SWORD_MOBILE - WP
      O "A-DBVALVES".ST7R.SWORD_MOBILE.test.fp_WP;
      = "A-DBVALVES".ST7R.SWORD_MOBILE.in.move_wp;

// Interlock wp
      L 0;
      T "A-DBVALVES".io[47].interlock_wp;

//{INTERLOCK_WP47}

      A(;
      L "A-DBVALVES".io[47].interlock_wp;
      L 0;
      <>I;
      );
      = "A-DBVALVES".ST7R.SWORD_MOBILE.interlock.wp_active;
NETWORK
TITLE = [47] ST7R MIECZ_RUCHOMY - IDLE
//[47] ST7R SWORD_MOBILE - IDLE
      O "A-DBVALVES".ST7R.SWORD_MOBILE.test.fp_IDLE;
      = "A-DBVALVES".ST7R.SWORD_MOBILE.in.move_idle;

// Interlock idle
      L 0;
      T "A-DBVALVES".io[47].interlock_idle;

//{INTERLOCK_IDLE47}

      A(;
      L "A-DBVALVES".io[47].interlock_idle;
      L 0;
      <>I;
      );
      = "A-DBVALVES".ST7R.SWORD_MOBILE.interlock.idle_active;
NETWORK
TITLE = [47] ST7R MIECZ_RUCHOMY
//[47] ST7R SWORD_MOBILE
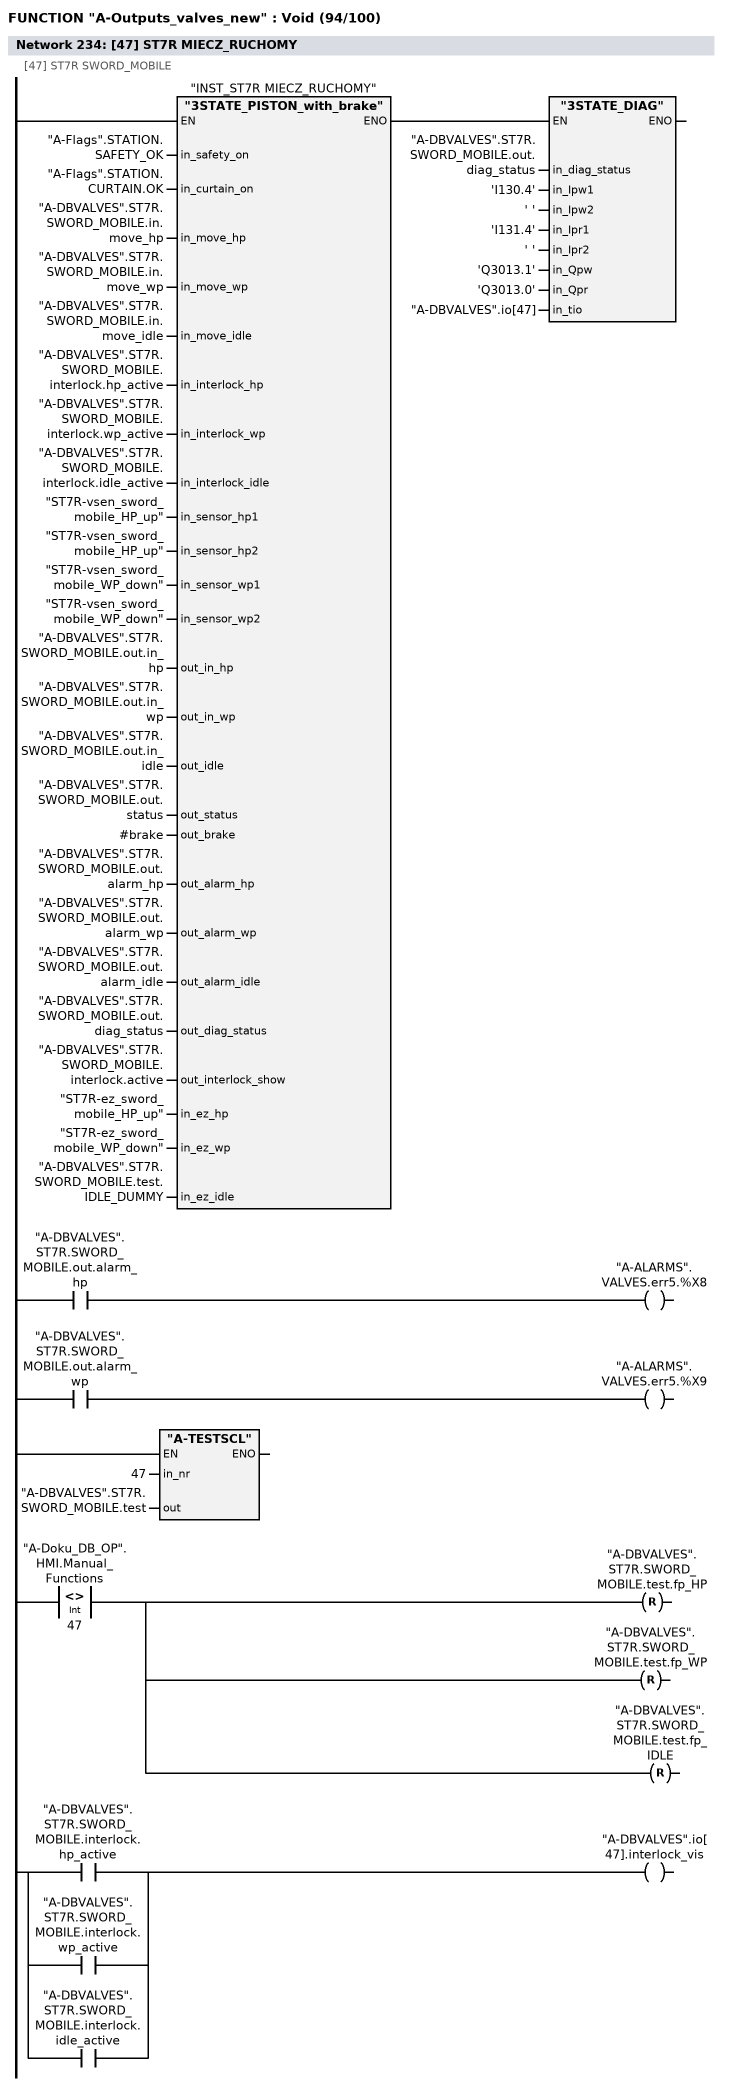
      CALL "3STATE_PISTON_with_brake", "INST_ST7R MIECZ_RUCHOMY"
      (  in_safety_on                := "A-Flags".STATION.SAFETY_OK ,
         in_curtain_on               := "A-Flags".STATION.CURTAIN.OK ,
         in_move_hp                  := "A-DBVALVES".ST7R.SWORD_MOBILE.in.move_hp ,
         in_move_wp                  := "A-DBVALVES".ST7R.SWORD_MOBILE.in.move_wp ,
         in_move_idle                := "A-DBVALVES".ST7R.SWORD_MOBILE.in.move_idle ,
         in_interlock_hp             := "A-DBVALVES".ST7R.SWORD_MOBILE.interlock.hp_active ,
         in_interlock_wp             := "A-DBVALVES".ST7R.SWORD_MOBILE.interlock.wp_active ,
         in_interlock_idle           := "A-DBVALVES".ST7R.SWORD_MOBILE.interlock.idle_active ,
         in_sensor_hp1               := "ST7R-vsen_sword_mobile_HP_up" ,
         in_sensor_hp2               := "ST7R-vsen_sword_mobile_HP_up" ,
         in_sensor_wp1               := "ST7R-vsen_sword_mobile_WP_down" ,
         in_sensor_wp2               := "ST7R-vsen_sword_mobile_WP_down" ,
         out_in_hp                   := "A-DBVALVES".ST7R.SWORD_MOBILE.out.in_hp ,
         out_in_wp                   := "A-DBVALVES".ST7R.SWORD_MOBILE.out.in_wp ,
         out_idle                    := "A-DBVALVES".ST7R.SWORD_MOBILE.out.in_idle ,
         out_status                  := "A-DBVALVES".ST7R.SWORD_MOBILE.out.status ,
         out_brake                   := #brake ,
         out_alarm_hp                := "A-DBVALVES".ST7R.SWORD_MOBILE.out.alarm_hp ,
         out_alarm_wp                := "A-DBVALVES".ST7R.SWORD_MOBILE.out.alarm_wp ,
         out_alarm_idle              := "A-DBVALVES".ST7R.SWORD_MOBILE.out.alarm_idle ,
         out_diag_status             := "A-DBVALVES".ST7R.SWORD_MOBILE.out.diag_status ,
         out_interlock_show          := "A-DBVALVES".ST7R.SWORD_MOBILE.interlock.active ,
         in_ez_hp                    := "ST7R-ez_sword_mobile_HP_up" ,
         in_ez_wp                    := "ST7R-ez_sword_mobile_WP_down" ,
         in_ez_idle                  := "A-DBVALVES".ST7R.SWORD_MOBILE.test.IDLE_DUMMY
      );

      CALL "3STATE_DIAG"
      (  in_diag_status              := "A-DBVALVES".ST7R.SWORD_MOBILE.out.diag_status ,
         in_Ipw1                     := 'I130.4' ,
         in_Ipw2                     := ' ' ,
         in_Ipr1                     := 'I131.4' ,
         in_Ipr2                     := ' ' ,
         in_Qpw                      := 'Q3013.1' ,
         in_Qpr                      := 'Q3013.0' ,
         in_tio                      := "A-DBVALVES".io[47]
      );

      A "A-DBVALVES".ST7R.SWORD_MOBILE.out.alarm_hp;
      = "A-ALARMS".VALVES.err5.%X8;

      A "A-DBVALVES".ST7R.SWORD_MOBILE.out.alarm_wp;
      = "A-ALARMS".VALVES.err5.%X9;

      CALL "A-TESTSCL"
      (  in_nr                       := 47 ,
         out                         := "A-DBVALVES".ST7R.SWORD_MOBILE.test
      );

      A(;
      L "A-Doku_DB_OP".HMI.Manual_Functions;
      L 47;
      <>I;
      );
      R "A-DBVALVES".ST7R.SWORD_MOBILE.test.fp_HP;
      R "A-DBVALVES".ST7R.SWORD_MOBILE.test.fp_WP;
      R "A-DBVALVES".ST7R.SWORD_MOBILE.test.fp_IDLE;

      O "A-DBVALVES".ST7R.SWORD_MOBILE.interlock.hp_active;
      O "A-DBVALVES".ST7R.SWORD_MOBILE.interlock.wp_active;
      O "A-DBVALVES".ST7R.SWORD_MOBILE.interlock.idle_active;
      = "A-DBVALVES".io[47].interlock_vis;
NETWORK
TITLE = -

NETWORK
TITLE = [48] ST7 DOCISK_DOJAZD - HP
//[48] ST7 HOLDFAST_MOVEMENT - HP
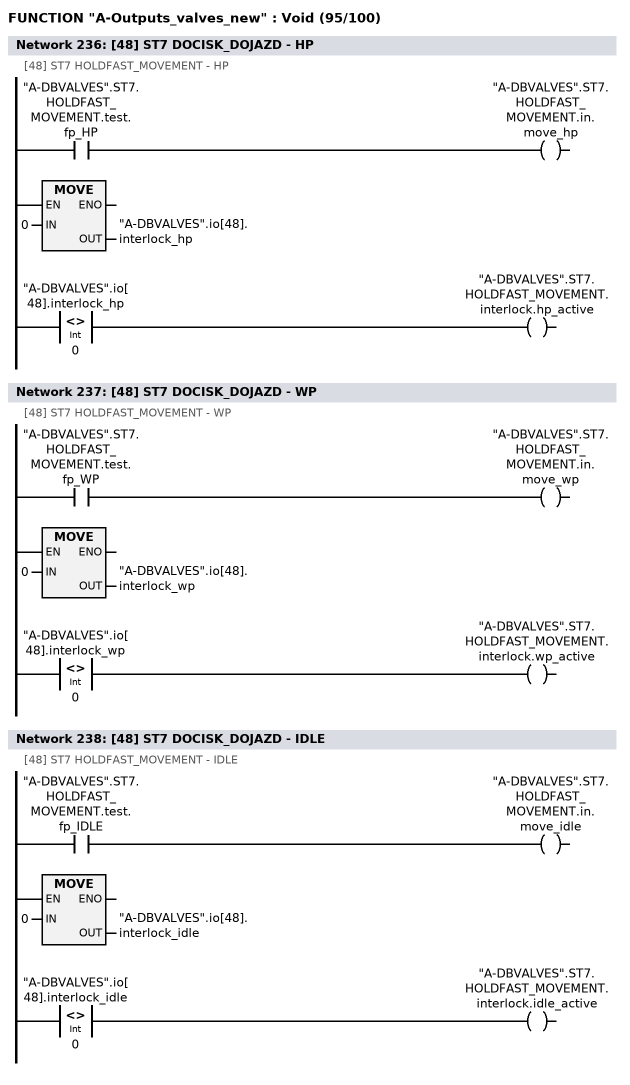
      O "A-DBVALVES".ST7.HOLDFAST_MOVEMENT.test.fp_HP;
//    O     "A-Flags".STATION.IN_HP_STEP
      = "A-DBVALVES".ST7.HOLDFAST_MOVEMENT.in.move_hp;

// Interlock hp
      L 0;
      T "A-DBVALVES".io[48].interlock_hp;

//{INTERLOCK_HP48}

      A(;
      L "A-DBVALVES".io[48].interlock_hp;
      L 0;
      <>I;
      );
      = "A-DBVALVES".ST7.HOLDFAST_MOVEMENT.interlock.hp_active;
NETWORK
TITLE = [48] ST7 DOCISK_DOJAZD - WP
//[48] ST7 HOLDFAST_MOVEMENT - WP
      O "A-DBVALVES".ST7.HOLDFAST_MOVEMENT.test.fp_WP;
      = "A-DBVALVES".ST7.HOLDFAST_MOVEMENT.in.move_wp;

// Interlock wp
      L 0;
      T "A-DBVALVES".io[48].interlock_wp;

//{INTERLOCK_WP48}

      A(;
      L "A-DBVALVES".io[48].interlock_wp;
      L 0;
      <>I;
      );
      = "A-DBVALVES".ST7.HOLDFAST_MOVEMENT.interlock.wp_active;
NETWORK
TITLE = [48] ST7 DOCISK_DOJAZD - IDLE
//[48] ST7 HOLDFAST_MOVEMENT - IDLE
      O "A-DBVALVES".ST7.HOLDFAST_MOVEMENT.test.fp_IDLE;
      = "A-DBVALVES".ST7.HOLDFAST_MOVEMENT.in.move_idle;

// Interlock idle
      L 0;
      T "A-DBVALVES".io[48].interlock_idle;

//{INTERLOCK_IDLE48}

      A(;
      L "A-DBVALVES".io[48].interlock_idle;
      L 0;
      <>I;
      );
      = "A-DBVALVES".ST7.HOLDFAST_MOVEMENT.interlock.idle_active;
NETWORK
TITLE = [48] ST7 DOCISK_DOJAZD
//[48] ST7 HOLDFAST_MOVEMENT
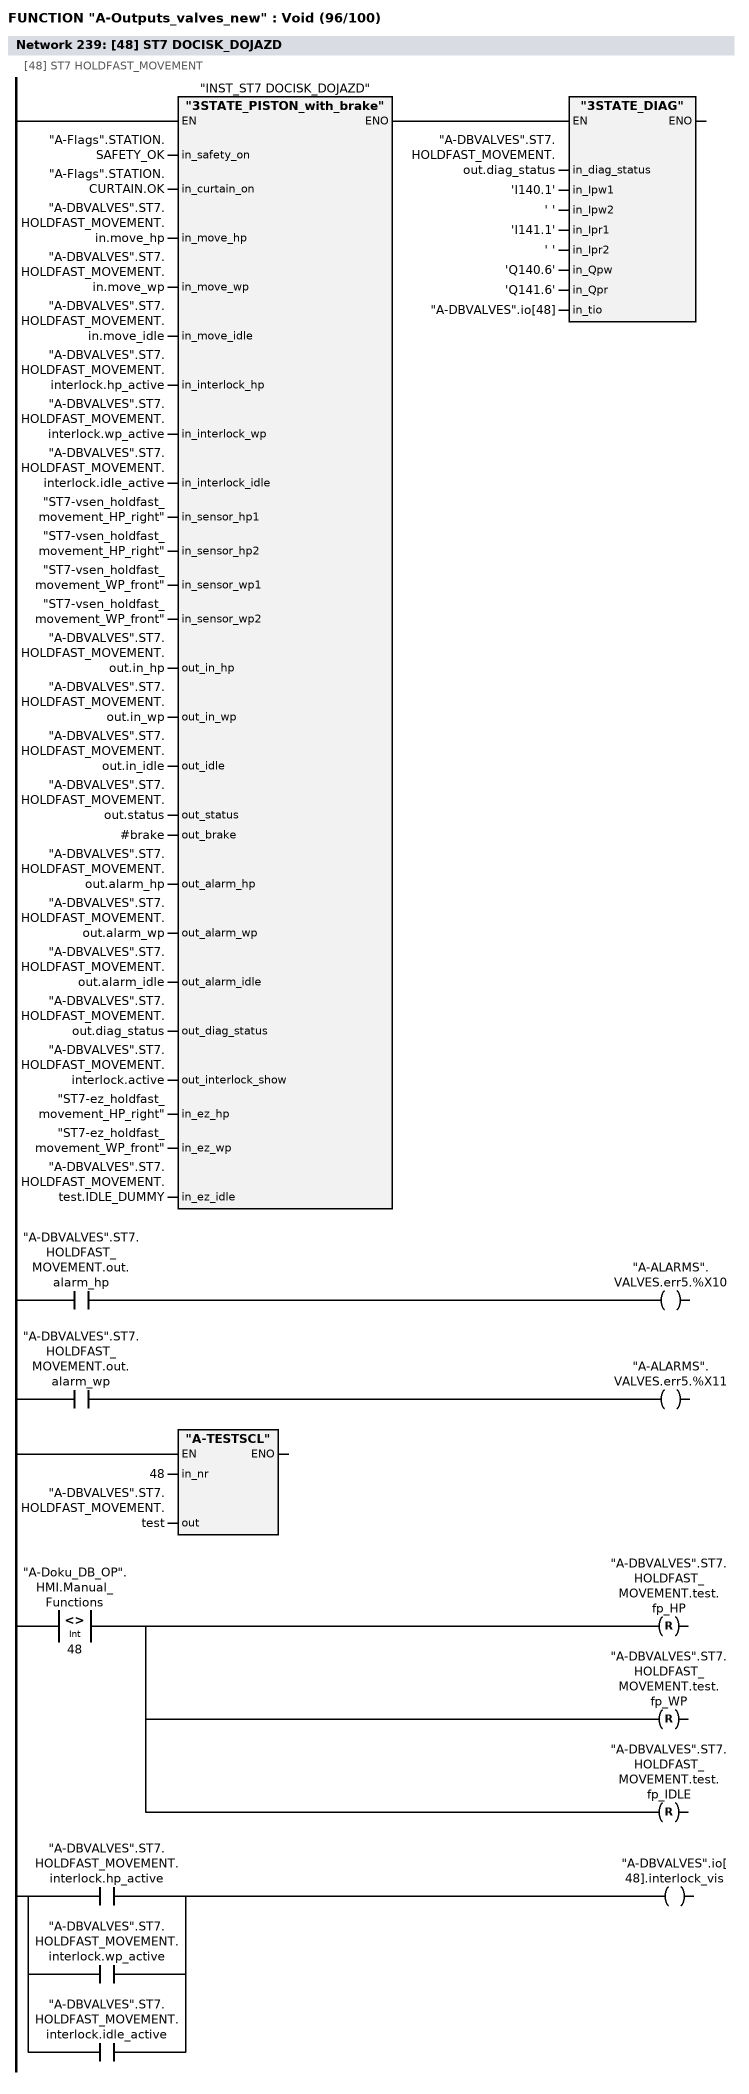
      CALL "3STATE_PISTON_with_brake", "INST_ST7 DOCISK_DOJAZD"
      (  in_safety_on                := "A-Flags".STATION.SAFETY_OK ,
         in_curtain_on               := "A-Flags".STATION.CURTAIN.OK ,
         in_move_hp                  := "A-DBVALVES".ST7.HOLDFAST_MOVEMENT.in.move_hp ,
         in_move_wp                  := "A-DBVALVES".ST7.HOLDFAST_MOVEMENT.in.move_wp ,
         in_move_idle                := "A-DBVALVES".ST7.HOLDFAST_MOVEMENT.in.move_idle ,
         in_interlock_hp             := "A-DBVALVES".ST7.HOLDFAST_MOVEMENT.interlock.hp_active ,
         in_interlock_wp             := "A-DBVALVES".ST7.HOLDFAST_MOVEMENT.interlock.wp_active ,
         in_interlock_idle           := "A-DBVALVES".ST7.HOLDFAST_MOVEMENT.interlock.idle_active ,
         in_sensor_hp1               := "ST7-vsen_holdfast_movement_HP_right" ,
         in_sensor_hp2               := "ST7-vsen_holdfast_movement_HP_right" ,
         in_sensor_wp1               := "ST7-vsen_holdfast_movement_WP_front" ,
         in_sensor_wp2               := "ST7-vsen_holdfast_movement_WP_front" ,
         out_in_hp                   := "A-DBVALVES".ST7.HOLDFAST_MOVEMENT.out.in_hp ,
         out_in_wp                   := "A-DBVALVES".ST7.HOLDFAST_MOVEMENT.out.in_wp ,
         out_idle                    := "A-DBVALVES".ST7.HOLDFAST_MOVEMENT.out.in_idle ,
         out_status                  := "A-DBVALVES".ST7.HOLDFAST_MOVEMENT.out.status ,
         out_brake                   := #brake ,
         out_alarm_hp                := "A-DBVALVES".ST7.HOLDFAST_MOVEMENT.out.alarm_hp ,
         out_alarm_wp                := "A-DBVALVES".ST7.HOLDFAST_MOVEMENT.out.alarm_wp ,
         out_alarm_idle              := "A-DBVALVES".ST7.HOLDFAST_MOVEMENT.out.alarm_idle ,
         out_diag_status             := "A-DBVALVES".ST7.HOLDFAST_MOVEMENT.out.diag_status ,
         out_interlock_show          := "A-DBVALVES".ST7.HOLDFAST_MOVEMENT.interlock.active ,
         in_ez_hp                    := "ST7-ez_holdfast_movement_HP_right" ,
         in_ez_wp                    := "ST7-ez_holdfast_movement_WP_front" ,
         in_ez_idle                  := "A-DBVALVES".ST7.HOLDFAST_MOVEMENT.test.IDLE_DUMMY
      );

      CALL "3STATE_DIAG"
      (  in_diag_status              := "A-DBVALVES".ST7.HOLDFAST_MOVEMENT.out.diag_status ,
         in_Ipw1                     := 'I140.1' ,
         in_Ipw2                     := ' ' ,
         in_Ipr1                     := 'I141.1' ,
         in_Ipr2                     := ' ' ,
         in_Qpw                      := 'Q140.6' ,
         in_Qpr                      := 'Q141.6' ,
         in_tio                      := "A-DBVALVES".io[48]
      );

      A "A-DBVALVES".ST7.HOLDFAST_MOVEMENT.out.alarm_hp;
      = "A-ALARMS".VALVES.err5.%X10;

      A "A-DBVALVES".ST7.HOLDFAST_MOVEMENT.out.alarm_wp;
      = "A-ALARMS".VALVES.err5.%X11;

      CALL "A-TESTSCL"
      (  in_nr                       := 48 ,
         out                         := "A-DBVALVES".ST7.HOLDFAST_MOVEMENT.test
      );

      A(;
      L "A-Doku_DB_OP".HMI.Manual_Functions;
      L 48;
      <>I;
      );
      R "A-DBVALVES".ST7.HOLDFAST_MOVEMENT.test.fp_HP;
      R "A-DBVALVES".ST7.HOLDFAST_MOVEMENT.test.fp_WP;
      R "A-DBVALVES".ST7.HOLDFAST_MOVEMENT.test.fp_IDLE;

      O "A-DBVALVES".ST7.HOLDFAST_MOVEMENT.interlock.hp_active;
      O "A-DBVALVES".ST7.HOLDFAST_MOVEMENT.interlock.wp_active;
      O "A-DBVALVES".ST7.HOLDFAST_MOVEMENT.interlock.idle_active;
      = "A-DBVALVES".io[48].interlock_vis;
NETWORK
TITLE = -

NETWORK
TITLE = [49] ST7 DOCISK_WYSUW - HP
//[49] ST7 HOLDFAST_SLIDE_OUT - HP
